// TIA Portal V16 program export: 3 tag tables, 15 data types, 4 data blocks, 30 code blocks (in call order from the OBs), 9 instance data blocks

VAR_GLOBAL   // PLC tag table "Default tag table"
   System_Byte AT %MB1 : Byte;
   FirstScan AT %M1.0 : Bool;
   DiagStatusUpdate AT %M1.1 : Bool;
   AlwaysTRUE AT %M1.2 : Bool;
   AlwaysFALSE AT %M1.3 : Bool;
   Clock_Byte AT %MB0 : Byte;
   Clock_10Hz AT %M0.0 : Bool;
   Clock_5Hz AT %M0.1 : Bool;
   "Clock_2.5Hz" AT %M0.2 : Bool;
   Clock_2Hz AT %M0.3 : Bool;
   "Clock_1.25Hz" AT %M0.4 : Bool;
   Clock_1Hz AT %M0.5 : Bool;
   "Clock_0.625Hz" AT %M0.6 : Bool;
   "Clock_0.5Hz" AT %M0.7 : Bool;
   Tag_1 AT %M100.0 : Bool;
   Tag_2 AT %MW200 : Int;
   Tag_3 AT %M100.1 : Bool;
   Tag_4 AT %M100.2 : Bool;
   Tag_5 AT %M100.3 : Bool;
   Tag_6 AT %M100.4 : Bool;
   Tag_7 AT %M100.5 : Bool;
   Tag_8 AT %M200.0 : Bool;
   Tag_9 AT %MD300 : Real;
   pulse_high AT %M110.0 : Bool;
END_VAR

VAR_GLOBAL   // PLC tag table "input"
   buttonControlCircuit AT %I0.0 : Bool;   // цепи управления
   buttonStart AT %I0.1 : Bool;   // Старт
   buttonStop AT %I0.2 : Bool;   // Стоп
   buttonAlarmStop AT %I0.3 : Bool;   // Аварийный стоп
   M1_alarmCB AT %I0.4 : Bool;   // М1 - авария автоматического выключателя
   M2_alarmCB AT %I0.5 : Bool;   // М2 - авария автоматического выключателя
   isNormalElectrical AT %I0.6 : Bool;   // Сеть в норме
   sensorOverflowReceiverTable AT %I0.7 : Bool;   // Датчик пересыпа приемного стола
   YP1_ReadyAccept AT %I1.0 : Bool;   // УП1 - готов принять
   YP1_StartDozing AT %I1.1 : Bool;   // УП1 - запуск дозирования
   YP2_ReadyAccept AT %I1.2 : Bool;   // УП2 - готов принять
   YP2_StartDozing AT %I1.3 : Bool;   // УП2 - запуск дозирования
END_VAR

VAR_GLOBAL   // PLC tag table "output"
   lampBlue AT %Q0.0 : Bool;   // Синяя лампа
   lampGreen AT %Q0.1 : Bool;   // Зеленая лампа
   lampRed AT %Q0.2 : Bool;   // Красная лампа
   qOn_ControlCurcuit AT %Q0.3 : Bool;   // включение цепей управления
   Y1q_ReadyDoze AT %Q0.4 : Bool;   // УП1 - доза готова
   Y2q_ReadyDoze AT %Q0.5 : Bool;   // УП2 - доза готова
   Conv1_FRV AT %Q0.6 : Bool;   // Конвейер1 - вперед
   Conv1_REV AT %Q0.7 : Bool;   // Конвейер1 - назад
   Conv2_FRV AT %Q1.0 : Bool;   // Конвейер2 - вперед
   Conv2_REV AT %Q1.1 : Bool;   // Конвейер2 - назад
   qDoor1_open AT %Q8.0 : Bool;   // Лопатка - открыть - 1
   qDoor1_close AT %Q8.1 : Bool;   // Лопатка - закрыть- 1
   qDoor2_open AT %Q8.2 : Bool;   // Лопатка - открыть - 2
   qDoor2_close AT %Q8.3 : Bool;   // Лопатка - закрыть- 2
   qDoor3_open AT %Q8.4 : Bool;   // Лопатка - открыть - 3
   qDoor3_close AT %Q8.5 : Bool;   // Лопатка - закрыть- 3
   qDoor4_open AT %Q8.6 : Bool;   // Лопатка - открыть - 4
   qDoor4_close AT %Q8.7 : Bool;   // Лопатка - закрыть- 4
   qDoor5_open AT %Q9.0 : Bool;   // Лопатка - открыть - 5
   qDoor5_close AT %Q9.1 : Bool;   // Лопатка - закрыть- 5
   qDoor6_open AT %Q9.2 : Bool;   // Лопатка - открыть - 6
   qDoor6_close AT %Q9.3 : Bool;   // Лопатка - закрыть- 6
   qDoor7_open AT %Q9.4 : Bool;   // Лопатка - открыть - 7
   qDoor7_close AT %Q9.5 : Bool;   // Лопатка - закрыть- 7
   qDoor8_open AT %Q9.6 : Bool;   // Лопатка - открыть - 8
   qDoor8_close AT %Q9.7 : Bool;   // Лопатка - закрыть- 8
   qBunker3_leftOpen AT %Q12.0 : Bool;   // Бункер - открыть влево - 3
   qBunker3_leftClose AT %Q12.1 : Bool;   // Бункер - закрыть влево - 3
   qBunker3_rightOpen AT %Q12.2 : Bool;   // Бункер - открыть вправо- 3
   qBunker3_rightClose AT %Q12.3 : Bool;   // Бункер - закрыть вправо- 3
   qBunker4_leftOpen AT %Q12.4 : Bool;   // Бункер - открыть влево - 4
   qBunker4_leftClose AT %Q12.5 : Bool;   // Бункер - закрыть влево - 4
   qBunker4_rightOpen AT %Q12.6 : Bool;   // Бункер - открыть вправо- 4
   qBunker4_rightClose AT %Q12.7 : Bool;   // Бункер - закрыть вправо- 4
   qBunker5_leftOpen AT %Q13.0 : Bool;   // Бункер - открыть влево - 5
   qBunker5_leftClose AT %Q13.1 : Bool;   // Бункер - закрыть влево - 5
   qBunker5_rightOpen AT %Q13.2 : Bool;   // Бункер - открыть вправо- 5
   qBunker5_rightClose AT %Q13.3 : Bool;   // Бункер - закрыть вправо- 5
   qBunker6_leftOpen AT %Q13.4 : Bool;   // Бункер - открыть влево - 6
   qBunker6_leftClose AT %Q13.5 : Bool;   // Бункер - закрыть влево - 6
   qBunker6_rightOpen AT %Q13.6 : Bool;   // Бункер - открыть вправо- 6
   qBunker6_rightClose AT %Q13.7 : Bool;   // Бункер - закрыть вправо- 6
   qBunker7_leftOpen AT %Q14.0 : Bool;   // Бункер - открыть влево - 7
   qBunker7_leftClose AT %Q14.1 : Bool;   // Бункер - закрыть влево - 7
   qBunker7_rightOpen AT %Q14.2 : Bool;   // Бункер - открыть вправо- 7
   qBunker7_rightClose AT %Q14.3 : Bool;   // Бункер - закрыть вправо- 7
   qBunker8_leftOpen AT %Q14.4 : Bool;   // Бункер - открыть влево - 8
   qBunker8_leftClose AT %Q14.5 : Bool;   // Бункер - закрыть влево - 8
   qBunker8_rightOpen AT %Q14.6 : Bool;   // Бункер - открыть вправо- 8
   qBunker8_rightClose AT %Q14.7 : Bool;   // Бункер - закрыть вправо- 8
   qBunker9_leftOpen AT %Q15.0 : Bool;   // Бункер - открыть влево - 9
   qBunker9_leftClose AT %Q15.1 : Bool;   // Бункер - закрыть влево - 9
   qBunker9_rightOpen AT %Q15.2 : Bool;   // Бункер - открыть вправо- 9
   qBunker9_rightClose AT %Q15.3 : Bool;   // Бункер - закрыть вправо- 9
   setVibration AT %QW64 : Int;   // задание уровня вибрации
   qDoor9_open AT %Q10.0 : Bool;   // Лопатка - открыть - 9
   qDoor9_close AT %Q10.1 : Bool;   // Лопатка - закрыть- 9
   qDoor10_open AT %Q10.2 : Bool;   // Лопатка - открыть - 10
   qDoor10_close AT %Q10.3 : Bool;   // Лопатка - закрыть- 10
   qDoor11_open AT %Q10.4 : Bool;   // Лопатка - открыть - 11
   qDoor11_close AT %Q10.5 : Bool;   // Лопатка - закрыть- 11
   qDoor12_open AT %Q10.6 : Bool;   // Лопатка - открыть - 12
   qDoor12_close AT %Q10.7 : Bool;   // Лопатка - закрыть- 12
   qBunker1_leftOpen AT %Q11.0 : Bool;   // Бункер - открыть влево - 1
   qBunker1_leftClose AT %Q11.1 : Bool;   // Бункер - закрыть влево - 1
   qBunker1_rightOpen AT %Q11.2 : Bool;   // Бункер - открыть вправо - 1
   qBunker1_rightClose AT %Q11.3 : Bool;   // Бункер - закрыть вправо - 1
   qBunker2_leftOpen AT %Q11.4 : Bool;   // Бункер - открыть влево - 2
   qBunker2_leftClose AT %Q11.5 : Bool;   // Бункер - закрыть влево - 2
   qBunker2_rightOpen AT %Q11.6 : Bool;   // Бункер - открыть вправо - 2
   qBunker2_rightClose AT %Q11.7 : Bool;   // Бункер - закрыть вправо - 2
   qBunker11_leftOpen AT %Q16.0 : Bool;   // Бункер - открыть влево - 11
   qBunker11_leftClose AT %Q16.1 : Bool;   // Бункер - закрыть влево - 11
   qBunker11_rightOpen AT %Q16.2 : Bool;   // Бункер - открыть вправо- 11
   qBunker11_rightClose AT %Q16.3 : Bool;   // Бункер - закрыть вправо- 11
   qBunker12_leftOpen AT %Q16.4 : Bool;   // Бункер - открыть влево - 12
   qBunker12_leftClose AT %Q16.5 : Bool;   // Бункер - закрыть влево - 12
   qBunker12_rightOpen AT %Q16.6 : Bool;   // Бункер - открыть вправо- 12
   qBunker12_rightClose AT %Q16.7 : Bool;   // Бункер - закрыть вправо- 12
   qBunker10_leftOpen AT %Q15.4 : Bool;   // Бункер - открыть влево - 10
   qBunker10_leftClose AT %Q15.5 : Bool;   // Бункер - закрыть влево - 10
   qBunker10_rightOpen AT %Q15.6 : Bool;   // Бункер - открыть вправо- 10
   qBunker10_rightClose AT %Q15.7 : Bool;   // Бункер - закрыть вправо- 10
   qFlipperUp AT %Q17.0 : Bool;   // плавник поднять
   qFlipperDown AT %Q17.1 : Bool;   // плавник опустить
   qVibroLot7_On AT %Q18.2 : Bool;   // управление вибролотком 7
   qVibroLot8_On AT %Q18.3 : Bool;   // управление вибролотком 8
   qVibroLot9_On AT %Q18.4 : Bool;   // управление вибролотком 9
   qVibroLot10_On AT %Q18.5 : Bool;   // управление вибролотком 10
   qVibroLot11_On AT %Q18.6 : Bool;   // управление вибролотком 11
   qVibroLot12_On AT %Q18.7 : Bool;   // управление вибролотком 12
   qVibroLot6_On AT %Q18.1 : Bool;   // управление вибролотком 6
   qVibroLot5_On AT %Q18.0 : Bool;   // управление вибролотком 5
   qVibroLot1_On AT %Q17.4 : Bool;   // управление вибролотком 1
   qVibroLot2_On AT %Q17.5 : Bool;   // управление вибролотком 2
   qVibroLot3_On AT %Q17.6 : Bool;   // управление вибролотком 3
   qVibroLot4_On AT %Q17.7 : Bool;   // управление вибролотком 4
   qVibroTable1 AT %Q17.2 : Bool;   // управление вибростолом 1
   qVibrotable2 AT %Q17.3 : Bool;   // управление вибростолом 2
   setSpeedConv AT %QW66 : Int;   // задание скорости конвейера
   startSourceConveyer AT %Q19.0 : Bool;   // запуск питателя
END_VAR

TYPE "LineWeight"
// stored: IsFailsafeCompliant false
   STRUCT
      isVibroLotWork : Bool;   // работа вибролотка
      percentVibroLot : Int;   // текущая вибрация вибролотка
      stateValveAfterVibroLot : Bool;   // состояние закрылки после вибролотка
      stateLeftValveWeightPocket : Bool;   // состояние левого клапана открывающегося кармана
      stateRightValveWeightPocket : Bool;   // состояние правого клапана открывающегося кармана
      targetWeightPocket : Real;   // целевой вес кармана
      currentWeightPocket : Real;   // текущий вес в кармане
      manOpenValveAfterVibroLot : Bool;   // ручн - открыть лопатку
      manCloseValveAfterVibroLot : Bool;   // ручн - закрыть лопатку
      manOpenLeftValveWeightPocket : Bool;   // ручн -открыть левый карман
      manCloseLeftValveWeightPocket : Bool;   // ручн -закрыть левый карман
      manOpenRightValveWeightPocket : Bool;   // ручн - открыть правый карман
      manCloseRightValveWieghtPocket : Bool;   // ручн - закрыть правый карман
      manVibroLotStart : Bool;   // ручн - управление ПУСК\Стоп вибролотка
      begWeightModuleReady : Bool;   // начальный экран - готовность весоизмерительного модуля
   END_STRUCT;
END_TYPE

TYPE "ReadyWeight"
// stored: IsFailsafeCompliant false
   STRUCT
      ready1Machine : Bool;
      ready2Machine : Bool;
   END_STRUCT;
END_TYPE

TYPE "addedVibro"
// stored: IsFailsafeCompliant false
   STRUCT
      manStartVibroTable : Array[0..2] of Bool;   // запуск вибростола в ручном режиме
      manValueVibro : Int;   // величина вибрации в ручном режиме
      stateVibroTable : Array[0..2] of Bool;
   END_STRUCT;
END_TYPE

TYPE "alarmsPlant"
// stored: IsFailsafeCompliant false
   STRUCT
      bit : Array[0..83] of Bool;
   END_STRUCT;
END_TYPE

TYPE "calibrationModule"
// stored: IsFailsafeCompliant false
   STRUCT
      calib : Array[0..12] of Bool;
      tara : Array[0..12] of Bool;
      valReadyWModule : Int;   // +- величина готовности модуля
   END_STRUCT;
END_TYPE

TYPE "cleaningMode"
// stored: IsFailsafeCompliant false
   STRUCT
      allWeightModuleReady : Bool;   // Все весоизмерительные модули готовы
      pauseClean : Bool;   // пауза очистки
      progressClean : Int;   // прогресс очистки
      runClean : Bool;   // запуск очистки
      timeClean : Int;   // время очистки
   END_STRUCT;
END_TYPE

TYPE "dataStantion"
// stored: IsFailsafeCompliant false
   STRUCT
      numberDozInMin : Int;   // число доз в минуту
      numberDozInthisWeight : Int;   // полученное число доз заданной порции
      nuvberDozSmena : Int;   // число доз за смену
      currentPogreshn1 : Real;   // погрешность для текущей дозы 1 машины
      currentPogr2 : Real;   // погрешность для текущей дозы 2 машины
      maxPogr : Real;   // максимальная погрешность для порции
      isEmulation : Bool;
      emulStartDozing : Array[0..2] of Bool;
      emulReadyAccept : Array[0..2] of Bool;
   END_STRUCT;
END_TYPE

TYPE "dateTime"
// stored: IsFailsafeCompliant false
   STRUCT
      year : Int;
      month : Int;
      day : Int;
      hour : Int;
      minute : Int;
      second : Int;
   END_STRUCT;
END_TYPE

TYPE "mode"
// stored: IsFailsafeCompliant false
   STRUCT
      Yq_ReadyDoze : Array[0..2] of Bool;
      Conv_FRV : Array[0..2] of Bool;   // Конвейер1 - вперед
      Conv_REV : Array[0..2] of Bool;   // Конвейер1 - назад
      Door_open : Array[0..12] of Bool;   // Лопатка - открыть
      Door_close : Array[0..12] of Bool;   // Лопатка - закрыть
      Bunker_leftOpen : Array[0..12] of Bool;   // Бункер - открыть влево
      Bunker_leftClose : Array[0..12] of Bool;   // Бункер - закрыть влево
      Bunker_rightOpen : Array[0..12] of Bool;   // Бункер - открыть вправо
      Bunker_rightClose : Array[0..12] of Bool;   // Бункер - закрыть вправо
      flipper_Up : Bool;   // управление плавником вверх
      flipper_Down : Bool;   // управление плавником вниз
      vibroTable : Array[0..2] of Bool;   // управление вибростолом
      vibroLot : Array[0..12] of Bool;   // управление вибролотком
      setVibration : Real;   // уставка вибрации
      setSpeedInConv : Real;   // скорость питателя
      startInConv : Bool;   // запуск питателя
   END_STRUCT;
END_TYPE

TYPE "outConv"
// stored: IsFailsafeCompliant false
   STRUCT
      isUpInBegin : Bool;   // направление вращения для упаковки
      isUseInBegin : Bool;   // использовать ли конвейер для упаковки
      isUpInEnd : Bool;   // направления вращения при очистке
      setWeightPack : Real;   // вес упаковки
      currentWeightPack : Real;   // текущий вес упаковки
      currentErrorMeasure : Real;   // текущая погрешность
      isWorkConv : Bool;   // работа конвейера
      isAlarmConv : Bool;   // авария конвейера
      isReadyPackingMachine : Bool;   // сигнал готовности упаковочной машины
      isReadyDozaPackingMachine : Bool;   // сигнал доза упаковочной машины
      manStartOutConv : Bool;   // ручн - запуск конвейера
      stateConvInt : Int;   // состояние конвейера
      manIsUpConv : Bool;   // ручн - конв вперед\назад
   END_STRUCT;
END_TYPE

TYPE "plavnik"
// stored: IsFailsafeCompliant false
   STRUCT
      statePlavnik : Bool;   // состояние плавника
      manOpenPlavnik : Bool;   // ручн - открытие клапана
      manClosePlavnik : Bool;   // ручн - закрытие клапана
   END_STRUCT;
END_TYPE

TYPE "recipeVar"
// stored: IsFailsafeCompliant false
   STRUCT
      setWeight : Real;   // весовая уставка в рецепте
      speed_InConveyer : Int;   // скорость конвейера питателя( конвейер на входе системы)
      speedVibro : Int;   // скорость вибролотков(одна на все)
      maxWeightBunker : Real;   // максимальный вес бункеров
      workPlavnik : Bool;   // работа плавника
      measurmentError : Real;   // допускаемая погрешность веса в общем сбросе
      mediumWeightProduct : Real;   // средний вес продукта
   END_STRUCT;
END_TYPE

TYPE "rotary"
// stored: IsFailsafeCompliant false
   STRUCT
      rotUp1 : Int;
      rotDown1 : Int;
      rotUp2 : Int;
      rotDown2 : Int;
   END_STRUCT;
END_TYPE

TYPE "sourceConv"
// stored: IsFailsafeCompliant false
   STRUCT
      currentSpeed : Int;   // ОС скорость
      manSetSpeed : Int;   // ручн - задание скорости
      isConvWork : Bool;   // конв работает
      isConvAlarm : Bool;   // авария конв
      manStartConv : Bool;   // ручн - старт конвейера
      stateConvInt : Int;   // состояние конвейера
      setSpeedWeightLimit : Int;   // скорость питателя при перевесе
   END_STRUCT;
END_TYPE

TYPE "stableWeight"
// stored: IsFailsafeCompliant false
   STRUCT
      weight : Array[0..10] of Real;
   END_STRUCT;
END_TYPE

DATA_BLOCK "IO"   // DB10
{ S7_Optimized_Access := 'TRUE' }
VERSION : 0.1
// stored: AutoNumber false, DBAccessibleFromOPCUA true, IsOnlyStoredInLoadMemory false, IsRetainMemResEnabled false, IsWriteProtectedInAS false, MemoryReserve 100
   VAR
      input : Struct
         buttonControlCircuit : Bool;   // цепи управления
         buttonStart : Bool;   // Старт
         buttonStop : Bool;   // Стоп
         buttonAlarmStop : Bool;   // Аварийный стоп
         M_alarmCB : Array[0..2] of Bool;   // М - авария автоматического выключателя
         isNormalElectrical : Bool;   // Сеть в норме
         sensorOverflowReceiverTable : Bool;   // Датчик пересыпа приемного стола
         YP_ReadyAccept : Array[0..2] of Bool;   // УП - готов принять
         YP_StartDozing : Array[0..2] of Bool;   // УП - запуск дозирования
      END_STRUCT;
      output : Struct
         lampBlue : Bool;   // Синяя лампа
         lampGreen : Bool;   // Зеленая лампа
         lampRed : Bool;   // Красная лампа
         qOn_ControlCurcuit : Bool;   // включение цепей управления
         Yq_ReadyDoze : Array[0..2] of Bool;   // УП - доза готова
         Conv_FRV : Array[0..2] of Bool;   // Конвейер1 - вперед
         Conv_REV : Array[0..2] of Bool;   // Конвейер1 - назад
         Door_open : Array[0..12] of Bool;   // Лопатка - открыть
         Door_close : Array[0..12] of Bool;   // Лопатка - закрыть
         Bunker_leftOpen : Array[0..12] of Bool;   // Бункер - открыть влево
         Bunker_leftClose : Array[0..12] of Bool;   // Бункер - закрыть влево
         Bunker_rightOpen : Array[0..12] of Bool;   // Бункер - открыть вправо
         Bunker_rightClose : Array[0..12] of Bool;   // Бункер - закрыть вправо
         flipper_Up : Bool;   // управление плавником вверх
         flipper_Down : Bool;   // управление плавником вниз
         vibroTable : Array[0..2] of Bool;   // управление вибростолом
         vibroLot : Array[0..12] of Bool;   // управление вибролотком
         setVibration : Real;   // уставка вибрации
         setSpeed : Real;   // уставка скорости конвейера
         convSource : Bool;   // запуск питателя
      END_STRUCT;
   END_VAR
BEGIN
END_DATA_BLOCK

DATA_BLOCK "hmi"   // DB200
{ S7_Optimized_Access := 'FALSE' }
VERSION : 0.1
// stored: AutoNumber false, DBAccessibleFromOPCUA true, IsOnlyStoredInLoadMemory false, IsWriteProtectedInAS false
   VAR
      alarmTest : "alarmsPlant";
      autoMode : Bool;   // автоматический режим
      isEnableAutoMode : Bool;
      calibrWeightMode : "calibrationModule";   // калибровка и тарирование весов
      dataStantion : "dataStantion";
      manRunAllVibroLot : Bool;
      manStopAllVibroLot : Bool;
      NewReadyWeightOnLine : Array[0..12] of Bool;
      outConvAndPack : Array[0..2] of "outConv";
      permitOn1Bunk : Array[0..12] of Bool;
      permitOn2Bunk : Array[0..12] of Bool;
      plavnik : "plavnik";
      readySystem : Int;
      recipeVar : "recipeVar";   // переменные рецепта
      rotary : "rotary";   // анимация вращения конвейеров
      sourceConv : "sourceConv";
      timeWorkConvAuto : Int;
      weightLine : Array[0..12] of "LineWeight";
      currentSetRecipes : String := '$00$00';
      numPage : Int;
      commonAlarm : Bool;   // Сигнал если хотябы одна авария есть
      report : Struct
         perfomance : Int;   // производительность
         sumPreWeight : Real;   // суммарная переработка веса
         commonTimeWork : Real;   // время работы установки
      END_STRUCT;
      addedVibro : "addedVibro";
   END_VAR
BEGIN
   // alarmTest.bit[0] : Управляющие цепи деактивированны
   // alarmTest.bit[1] : весовой модуль не в сети 1
   // alarmTest.bit[2] : весовой модуль не в сети 2
   // alarmTest.bit[3] : весовой модуль не в сети 3
   // alarmTest.bit[4] : весовой модуль не в сети 4
   // alarmTest.bit[5] : весовой модуль не в сети 5
   // alarmTest.bit[6] : весовой модуль не в сети 6
   // alarmTest.bit[7] : весовой модуль не в сети 7
   // alarmTest.bit[8] : весовой модуль не в сети 8
   // alarmTest.bit[9] : весовой модуль не в сети 9
   // alarmTest.bit[10] : весовой модуль не в сети 10
   // alarmTest.bit[11] : весовой модуль не в сети 11
   // alarmTest.bit[12] : весовой модуль не в сети 12
   // alarmTest.bit[13] : обрыв датчик весового модуля 1 -значение выше 7000
   // alarmTest.bit[14] : обрыв датчик весового модуля 2
   // alarmTest.bit[15] : обрыв датчик весового модуля 3
   // alarmTest.bit[16] : обрыв датчик весового модуля 4
   // alarmTest.bit[17] : обрыв датчик весового модуля 5
   // alarmTest.bit[18] : обрыв датчик весового модуля 6
   // alarmTest.bit[19] : обрыв датчик весового модуля 7
   // alarmTest.bit[20] : обрыв датчик весового модуля 8
   // alarmTest.bit[21] : обрыв датчик весового модуля 9
   // alarmTest.bit[22] : обрыв датчик весового модуля 10
   // alarmTest.bit[23] : обрыв датчик весового модуля 11
   // alarmTest.bit[24] : обрыв датчик весового модуля 12
   // alarmTest.bit[25] : Напряжение сети не в норме
   // alarmTest.bit[26] : Тепловое реле Конв1
   // alarmTest.bit[27] : тепловое реле Конв2
   // alarmTest.bit[58] : Нажат аварийный пост
   // alarmTest.bit[59] : Авария бункер 1
   // alarmTest.bit[60] : Авария бункер 2
   // alarmTest.bit[61] : Авария бункер 3
   // alarmTest.bit[62] : Авария бункер 4
   // alarmTest.bit[63] : Авария бункер 5
   // alarmTest.bit[64] : Авария бункер 6
   // alarmTest.bit[65] : Авария бункер 7
   // alarmTest.bit[66] : Авария бункер 8
   // alarmTest.bit[67] : Авария бункер 9
   // alarmTest.bit[68] : Авария бункер 10
   // alarmTest.bit[69] : Авария бункер 11
   // alarmTest.bit[70] : Авария бункер 12
   // alarmTest.bit[83] : Нет возможности сформировать порцию
   // calibrWeightMode.calib : калибровка весов
   // calibrWeightMode.tara : тарирование весов
END_DATA_BLOCK

DATA_BLOCK "signalKVSStation"   // DB20
{ S7_Optimized_Access := 'TRUE' }
VERSION : 0.1
// stored: AutoNumber false, DBAccessibleFromOPCUA true, IsOnlyStoredInLoadMemory false, IsRetainMemResEnabled false, IsWriteProtectedInAS false, MemoryReserve 100
   VAR
      isWorkControlCircuit : Bool;   // цепи управления активированы
      isStopAlarm : Bool;   // приход любой аварии которая останавливает установку
      isOtherAlarm : Bool;   // приход просто аварий
      isStartAutoMode : Bool;   // начало работы в автоматическом режиме
      enableAutoMode : Bool;   // разрешение перевода в автоматический режим
      isPreparationAutoModeFinish : Bool;   // подготовк к запуску автоматического режима
      enableManualMode : Bool;   // разрешение работы в ручном режиме
      qManualMode : "mode";   // активация катушек в ручном режиме
      qAutoMode : "mode";   // активация катушек в автоматическом режиме
      currentWeight : Array[0..12] of Real;   // вес получаемый по модбасу
      stableWeight : Array[0..12] of "stableWeight";   // установившийся вес в бункерах
   END_VAR
BEGIN
END_DATA_BLOCK

DATA_BLOCK "bufferModBus"   // DB4
{ S7_Optimized_Access := 'FALSE' }
VERSION : 0.1
// stored: AutoNumber true, DBAccessibleFromOPCUA true, IsOnlyStoredInLoadMemory false, IsWriteProtectedInAS false
   VAR
      Buffer_DataModbusPort1 { ExternalAccessible := 'False'; ExternalVisible := 'False'; ExternalWritable := 'False'} : Array[0..20] of Word;
      Buffer_DataModbusPort2 { ExternalAccessible := 'False'; ExternalVisible := 'False'; ExternalWritable := 'False'} : Array[0..20] of Word;
   END_VAR
BEGIN
END_DATA_BLOCK

ORGANIZATION_BLOCK "Main"   // OB1, LAD, ProgramCycle
TITLE = "Main Program Sweep (Cycle)"
{ S7_Optimized_Access := 'TRUE' }
VERSION : 0.1
// stored: AutoNumber true, IsIECCheckEnabled false, SetENOAutomatically false
   VAR_INPUT
      Initial_Call : Bool;   // Initial call of this OB
      Remanence : Bool;   // =True, if remanent data are available
   END_VAR
BEGIN

REGION Network 1: опрос весов
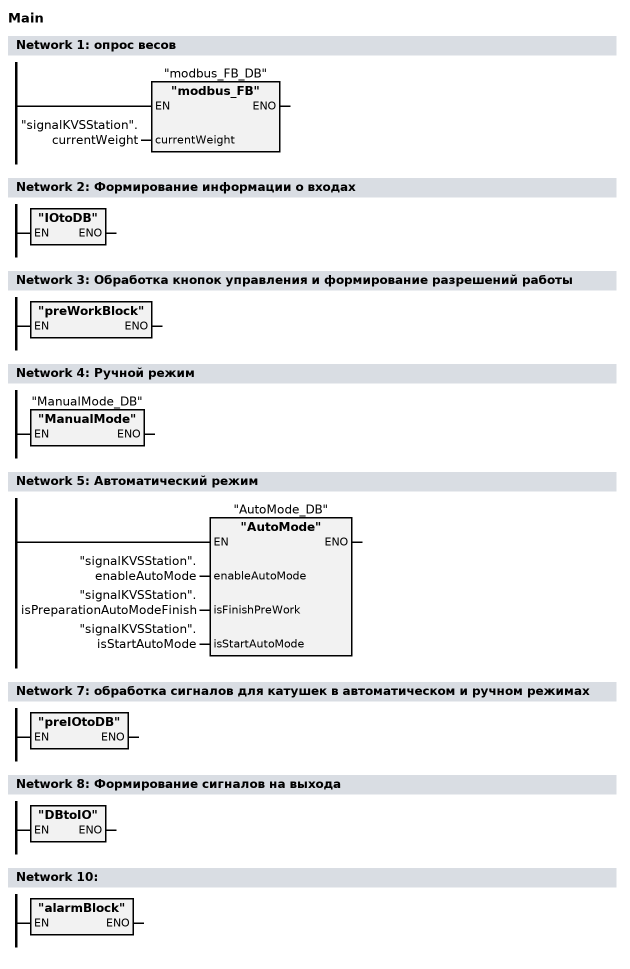
   RUNG wire#powerrail
      "modbus_FB_DB"(currentWeight := "signalKVSStation".currentWeight)
   END_RUNG
   // the same network as SCL:
   "modbus_FB_DB"(currentWeight := "signalKVSStation".currentWeight);   // "modbus_FB"
END_REGION

REGION Network 2: Формирование информации о входах
   RUNG wire#powerrail
      "IOtoDB"()
   END_RUNG
   // the same network as SCL:
   "IOtoDB"();
END_REGION

REGION Network 3: Обработка кнопок управления и формирование разрешений работы
   RUNG wire#powerrail
      "preWorkBlock"()
   END_RUNG
   // the same network as SCL:
   "preWorkBlock"();
END_REGION

REGION Network 4: Ручной режим
   RUNG wire#powerrail
      "ManualMode_DB"()
   END_RUNG
   // the same network as SCL:
   "ManualMode_DB"();   // "ManualMode"
END_REGION

REGION Network 5: Автоматический режим
   RUNG wire#powerrail
      "AutoMode_DB"(enableAutoMode := "signalKVSStation".enableAutoMode, isFinishPreWork := "signalKVSStation".isPreparationAutoModeFinish, isStartAutoMode := "signalKVSStation".isStartAutoMode)
   END_RUNG
   // the same network as SCL:
   "AutoMode_DB"(enableAutoMode := "signalKVSStation".enableAutoMode,   // "AutoMode"
                 isFinishPreWork := "signalKVSStation".isPreparationAutoModeFinish,
                 isStartAutoMode := "signalKVSStation".isStartAutoMode);
END_REGION

REGION Network 7: обработка сигналов для катушек в автоматическом и ручном режимах
   RUNG wire#powerrail
      "preIOtoDB"()
   END_RUNG
   // the same network as SCL:
   "preIOtoDB"();
END_REGION

REGION Network 8: Формирование сигналов на выхода
   RUNG wire#powerrail
      "DBtoIO"()
   END_RUNG
   // the same network as SCL:
   "DBtoIO"();
END_REGION

REGION Network 10
   RUNG wire#powerrail
      "alarmBlock"()
   END_RUNG
   // the same network as SCL:
   "alarmBlock"();
END_REGION
END_ORGANIZATION_BLOCK

FUNCTION_BLOCK "modbus_FB"   // FB9, LAD
{ S7_Optimized_Access := 'TRUE' }
VERSION : 0.1
// stored: AutoNumber true, IsIECCheckEnabled false, IsRetainMemResEnabled false, MemoryReserve 100, SetENOAutomatically false, UDAEnableTagReadback false
   VAR_IN_OUT
      currentWeight : Array[0..12] of Real;
   END_VAR
   VAR
      MODBUS_ADDRESS : Array[0..12] of UInt;
      modbus_SenecaConnectPort1_FB : "modbus_SenecaConnectPort1";
      modbus_SenecaConnectPort2_FB : "modbus_SenecaConnectPort2";
   END_VAR
   VAR_TEMP
      i : SInt;
   END_VAR
   // MODBUS_ADDRESS[1] := 10;
   // MODBUS_ADDRESS[2] := 11;
   // MODBUS_ADDRESS[3] := 12;
   // MODBUS_ADDRESS[4] := 13;
   // MODBUS_ADDRESS[5] := 14;
   // MODBUS_ADDRESS[6] := 15;
   // MODBUS_ADDRESS[7] := 20;
   // MODBUS_ADDRESS[8] := 21;
   // MODBUS_ADDRESS[9] := 22;
   // MODBUS_ADDRESS[10] := 23;
   // MODBUS_ADDRESS[11] := 24;
   // MODBUS_ADDRESS[12] := 25;
BEGIN

REGION Network 1: ОПРОС МОДУЛЕЙ ЧЕРЕРЗ 1 ПОРТ
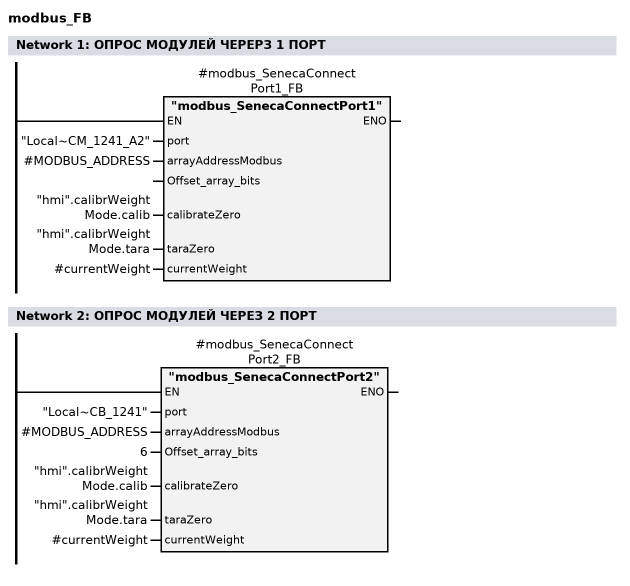
   RUNG wire#powerrail
      #modbus_SenecaConnectPort1_FB(port := "Local~CM_1241_A2", arrayAddressModbus := #MODBUS_ADDRESS, Offset_array_bits :=, calibrateZero := "hmi".calibrWeightMode.calib, taraZero := "hmi".calibrWeightMode.tara, currentWeight := #currentWeight)
   END_RUNG
   // the same network as SCL:
   #modbus_SenecaConnectPort1_FB(port := "Local~CM_1241_A2",   // "modbus_SenecaConnectPort1"
                           arrayAddressModbus := #MODBUS_ADDRESS,
                           calibrateZero := "hmi".calibrWeightMode.calib,
                           taraZero := "hmi".calibrWeightMode.tara,
                           currentWeight := #currentWeight);
END_REGION

REGION Network 2: ОПРОС МОДУЛЕЙ ЧЕРЕЗ 2 ПОРТ
   RUNG wire#powerrail
      #modbus_SenecaConnectPort2_FB(port := "Local~CB_1241", arrayAddressModbus := #MODBUS_ADDRESS, Offset_array_bits := 6, calibrateZero := "hmi".calibrWeightMode.calib, taraZero := "hmi".calibrWeightMode.tara, currentWeight := #currentWeight)
   END_RUNG
   // the same network as SCL:
   #modbus_SenecaConnectPort2_FB(port := "Local~CB_1241",   // "modbus_SenecaConnectPort2"
                           arrayAddressModbus := #MODBUS_ADDRESS,
                           Offset_array_bits := 6,
                           calibrateZero := "hmi".calibrWeightMode.calib,
                           taraZero := "hmi".calibrWeightMode.tara,
                           currentWeight := #currentWeight);
END_REGION

REGION Network 3 (SCL): Передаем вес в панель
   #i := 0;
   FOR #i := 1 TO 12 DO
       "hmi".weightLine[#i].currentWeightPocket := #currentWeight[#i];
   END_FOR;
END_REGION

REGION Network 4 (SCL)
   IF "hmi".calibrWeightMode.tara[0] THEN
       #i := 0;
       FOR #i := 1 TO 12 DO
           "hmi".calibrWeightMode.tara[#i] := true;
       END_FOR;
   END_IF;
END_REGION
END_FUNCTION_BLOCK

FUNCTION_BLOCK "modbus_SenecaConnectPort1"   // FB11, LAD
{ S7_Optimized_Access := 'TRUE' }
VERSION : 0.1
// stored: AutoNumber true, IsIECCheckEnabled false, IsRetainMemResEnabled false, MemoryReserve 100, SetENOAutomatically false, UDAEnableTagReadback false
   VAR_INPUT
      port : PORT;   // порт для подключения
      arrayAddressModbus : Array[0..12] of UInt;
      Offset_array_bits : SInt;
   END_VAR
   VAR_IN_OUT
      calibrateZero : Array[0..12] of Bool;
      taraZero : Array[0..12] of Bool;
      currentWeight : Array[0..12] of Real;
   END_VAR
   VAR
      MB_COMM_LOAD : MB_COMM_LOAD;
      MB_MASTER : MB_MASTER;
      Data_toMB_MASTER : Struct
         REQ : Bool;
         MB_ADDR : UInt;
         MODE : USInt;
         DATA_ADDR : UDInt;
         DATA_LEN : UInt;
         DONE : Bool;
         BUSY : Bool;
         ERROR : Bool;
      END_STRUCT;
      Seneca : Struct
         TON_changeStep : TON_TIME;
         TON_Start { S7_SetPoint := 'True'} : Bool;
         "Step" : SInt;
      END_STRUCT;
      tmpWeight : Array[0..12] of DWord;
      restartPort : Bool;   // перезагрузка Modbus
   END_VAR
   VAR_TEMP
      index : DInt;
      tmpIndex : DInt;
   END_VAR
   // MB_COMM_LOAD.RESP_TO := 100;
   VAR_TEMP   // added for the SCL form of the ladder/FBD networks
      _w1 : Bool;
   END_VAR
BEGIN

REGION Network 1: ИНИЦИАЛИЗИРУЕМ ПОРТ
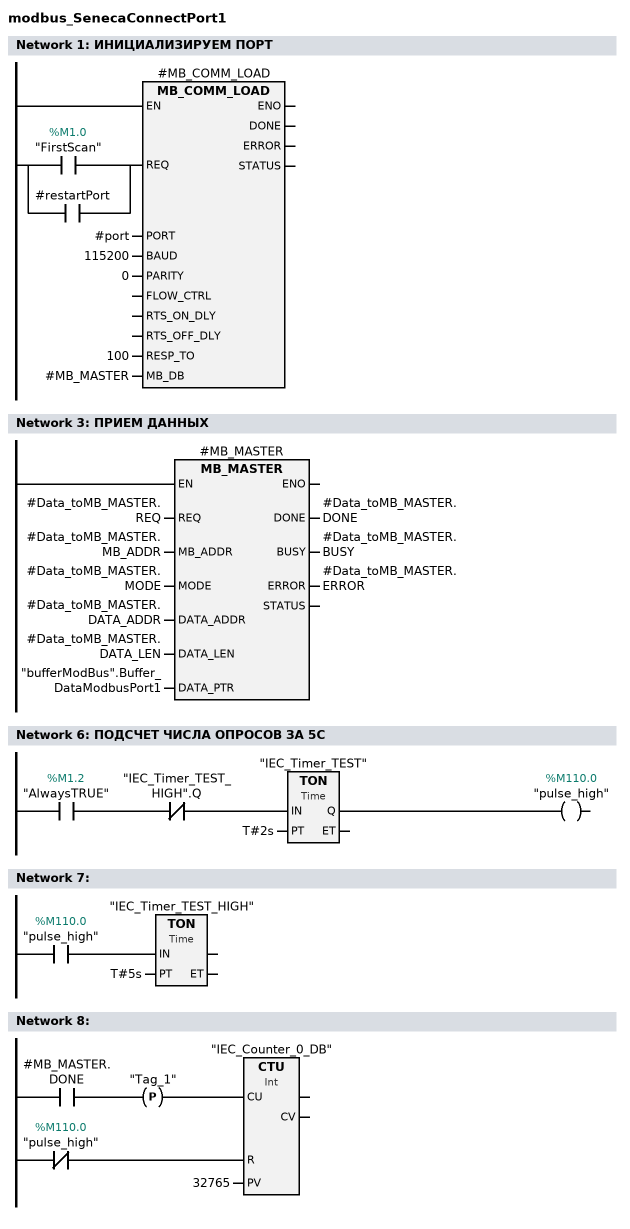
   RUNG wire#powerrail
      #MB_COMM_LOAD.MB_COMM_LOAD(REQ := wire#w1, PORT := #port, BAUD := 115200, PARITY := 0, FLOW_CTRL :=, RTS_ON_DLY :=, RTS_OFF_DLY :=, RESP_TO := 100, MB_DB := #MB_MASTER, DONE =>, ERROR =>, STATUS =>)
   END_RUNG
   RUNG wire#powerrail
      Contact( "FirstScan" )
   END_RUNG wire#w1
   RUNG wire#powerrail
      Contact( #restartPort )
   END_RUNG wire#w1
   // the same network as SCL:
   #MB_COMM_LOAD(REQ := "FirstScan" OR #restartPort,   // MB_COMM_LOAD
                 PORT := #port,
                 BAUD := 115200,
                 PARITY := 0,
                 RESP_TO := 100,
                 MB_DB := #MB_MASTER);
END_REGION

REGION Network 2 (SCL): ОБМЕН
   #Seneca.TON_changeStep(IN :=#Seneca.TON_Start,
                          PT := t#30ms);

   CASE #Seneca.Step OF

       1:
           #Seneca.Step := #Seneca.Step + 1;

       2: //ЧИТАЕМ ЗНАЧЕНИЕ ВЕСА С ПЕРВОГО МОДУЛЯ

           #index := 1+#Offset_array_bits;//заполнять функцию будем через индекс чтобы меньше писать
           "rcvDataWeight"(ADDR_DEVICE := #arrayAddressModbus[#index],
                           Ton_changeStep:=#Seneca.TON_changeStep.Q,
                           Ton_Start:=#Seneca.TON_Start,
                           "Step":=#Seneca.Step,
                           MB_MASTER:=#Data_toMB_MASTER);

       3://ЧИТАЕМ ЗНАЧЕНИЕ ВЕСА СО ВТОРОГО МОДУЛЯ
           #index := 2+#Offset_array_bits;//заполнять функцию будем через индекс чтобы меньше писать
           "rcvDataWeight"(ADDR_DEVICE := #arrayAddressModbus[#index],
                           Ton_changeStep:=#Seneca.TON_changeStep.Q,
                           Ton_Start:=#Seneca.TON_Start,
                           "Step":=#Seneca.Step,
                           MB_MASTER:=#Data_toMB_MASTER);

       4: // КАЛИБРОВКА 0 ДЛЯ ПЕРВОГО МОДУЛЯ и ТАРИРОВАНИЕ
           #index := 1+#Offset_array_bits;//заполнять функцию будем через индекс чтобы меньше писать
           "sndCALIBR&Tara"(ADDR_DEVICE := #arrayAddressModbus[#index],
                        ton_changeStep:=#Seneca.TON_changeStep.Q,
                        MB_MASTER:=#Data_toMB_MASTER,
                        Ton_Start:=#Seneca.TON_Start,
                        Calibrate:=#calibrateZero[#index],
                        Buffer:="bufferModBus".Buffer_DataModbusPort1,
                        "Step":=#Seneca.Step,
                        Tara:=#taraZero[#index]);


       5:// КАЛИБРОВКА 0 ДЛЯ ВТОРОГО МОДУЛЯ и ТАРИРОВАНИЕ
           #index := 2+#Offset_array_bits;//заполнять функцию будем через индекс чтобы меньше писать
           "sndCALIBR&Tara"(ADDR_DEVICE := #arrayAddressModbus[#index],
                        ton_changeStep := #Seneca.TON_changeStep.Q,
                        MB_MASTER := #Data_toMB_MASTER,
                        Ton_Start := #Seneca.TON_Start,
                        Calibrate := #calibrateZero[#index],
                        Buffer := "bufferModBus".Buffer_DataModbusPort1,
                        "Step" := #Seneca.Step,
                        Tara := #taraZero[#index]);

           //////////////////////////////////////////////////////////////////////////////////
           //////////////////////////////////////////////////////////////////////////////////
           //////////////////////////////////////////////////////////////////////////////////
           //////////////////////////////////////////////////////////////////////////////////
       6: //ЧИТАЕМ ЗНАЧЕНИЕ ВЕСА С ТРЕТЬЕГО МОДУЛЯ

           #index := 3+#Offset_array_bits;//заполнять функцию будем через индекс чтобы меньше писать
           "rcvDataWeight"(ADDR_DEVICE := #arrayAddressModbus[#index],
                           Ton_changeStep := #Seneca.TON_changeStep.Q,
                           Ton_Start := #Seneca.TON_Start,
                           "Step" := #Seneca.Step,
                           MB_MASTER := #Data_toMB_MASTER);

       7://ЧИТАЕМ ЗНАЧЕНИЕ ВЕСА С ЧЕТВЕРТОГО МОДУЛЯ
           #index := 4+#Offset_array_bits;//заполнять функцию будем через индекс чтобы меньше писать
           "rcvDataWeight"(ADDR_DEVICE := #arrayAddressModbus[#index],
                           Ton_changeStep := #Seneca.TON_changeStep.Q,
                           Ton_Start := #Seneca.TON_Start,
                           "Step" := #Seneca.Step,
                           MB_MASTER := #Data_toMB_MASTER);

       8:// КАЛИБРОВКА 0 ДЛЯ ТРЕТЬЕГО  МОДУЛЯ

           #index := 3+#Offset_array_bits;//заполнять функцию будем через индекс чтобы меньше писать
           "sndCALIBR&Tara"(ADDR_DEVICE := #arrayAddressModbus[#index],
                        ton_changeStep := #Seneca.TON_changeStep.Q,
                        MB_MASTER := #Data_toMB_MASTER,
                        Ton_Start := #Seneca.TON_Start,
                        Calibrate := #calibrateZero[#index],
                        Buffer := "bufferModBus".Buffer_DataModbusPort1,
                        "Step" := #Seneca.Step,
                        Tara := #taraZero[#index]);

       9://КАЛИБРОВКА 0 ДЛЯ ЧЕТВЕРТОГО МОДУЛЯ

           #index := 4+#Offset_array_bits;//заполнять функцию будем через индекс чтобы меньше писать
           "sndCALIBR&Tara"(ADDR_DEVICE := #arrayAddressModbus[#index],
                        ton_changeStep := #Seneca.TON_changeStep.Q,
                        MB_MASTER := #Data_toMB_MASTER,
                        Ton_Start := #Seneca.TON_Start,
                        Calibrate := #calibrateZero[#index],
                        Buffer := "bufferModBus".Buffer_DataModbusPort1,
                        "Step" := #Seneca.Step,
                        Tara := #taraZero[#index]);

           /////////////////////////////////////////////////////////////////////////////////
           ////////////////////////////////////////////////////////////////////////////////
           ////////////////////////////////////////////////////////////////////////////////
           ////////////////////////////////////////////////////////////////////////////////
       10: //ЧИТАЕМ ЗНАЧЕНИЕ ВЕСА С ПЯТОГО МОДУЛЯ
           #index := 5+#Offset_array_bits;//заполнять функцию будем через индекс чтобы меньше писать
           "rcvDataWeight"(ADDR_DEVICE := #arrayAddressModbus[#index],
                           Ton_changeStep := #Seneca.TON_changeStep.Q,
                           Ton_Start := #Seneca.TON_Start,
                           "Step" := #Seneca.Step,
                           MB_MASTER := #Data_toMB_MASTER);

       11://ЧИТАЕМ ЗНАЧЕНИЕ ВЕСА С ШЕСТОГО МОДУЛЯ
           #index := 6+#Offset_array_bits;//заполнять функцию будем через индекс чтобы меньше писать
           "rcvDataWeight"(ADDR_DEVICE := #arrayAddressModbus[#index],
                           Ton_changeStep := #Seneca.TON_changeStep.Q,
                           Ton_Start := #Seneca.TON_Start,
                           "Step" := #Seneca.Step,
                           MB_MASTER := #Data_toMB_MASTER);

       12:// КАЛИБРОВКА 0 ДЛЯ ПЯТОГО  МОДУЛЯ

           #index := 5+#Offset_array_bits;//заполнять функцию будем через индекс чтобы меньше писать
           "sndCALIBR&Tara"(ADDR_DEVICE := #arrayAddressModbus[#index],
                        ton_changeStep := #Seneca.TON_changeStep.Q,
                        MB_MASTER := #Data_toMB_MASTER,
                        Ton_Start := #Seneca.TON_Start,
                        Calibrate := #calibrateZero[#index],
                        Buffer := "bufferModBus".Buffer_DataModbusPort1,
                        "Step" := #Seneca.Step,
                        Tara := #taraZero[#index]);

       13:// КАЛИБРОВКА 0 ДЛЯ ШЕСТОГО МОДУЛЯ
           #index := 6+#Offset_array_bits;//заполнять функцию будем через индекс чтобы меньше писать
           "sndCALIBR&Tara"(ADDR_DEVICE := #arrayAddressModbus[#index],
                        ton_changeStep := #Seneca.TON_changeStep.Q,
                        MB_MASTER := #Data_toMB_MASTER,
                        Ton_Start := #Seneca.TON_Start,
                        Calibrate := #calibrateZero[#index],
                        Buffer := "bufferModBus".Buffer_DataModbusPort1,
                        "Step" := #Seneca.Step,
                        Tara := #taraZero[#index]);
   14://отправка аналоговых значений вибрации
       "sndVibration"(ADDR_DEVICE:=40,
                      ton_changeStep:= #Seneca.TON_changeStep.Q,
                      MB_MASTER:=#Data_toMB_MASTER,
                      Ton_Start:=#Seneca.TON_Start,
                      Buffer:="bufferModBus".Buffer_DataModbusPort1,
                      "Step":=#Seneca.Step);
   ELSE
           #Seneca.Step := 1;
   END_CASE;
END_REGION

REGION Network 3: ПРИЕМ ДАННЫХ
   RUNG wire#powerrail
      #MB_MASTER.MB_MASTER(REQ := #Data_toMB_MASTER.REQ, MB_ADDR := #Data_toMB_MASTER.MB_ADDR, MODE := #Data_toMB_MASTER.MODE, DATA_ADDR := #Data_toMB_MASTER.DATA_ADDR, DATA_LEN := #Data_toMB_MASTER.DATA_LEN, DATA_PTR := "bufferModBus".Buffer_DataModbusPort1, DONE => #Data_toMB_MASTER.DONE, BUSY => #Data_toMB_MASTER.BUSY, ERROR => #Data_toMB_MASTER.ERROR, STATUS =>)
   END_RUNG
   // the same network as SCL:
   #MB_MASTER(REQ := #Data_toMB_MASTER.REQ,   // MB_MASTER
              MB_ADDR := #Data_toMB_MASTER.MB_ADDR,
              MODE := #Data_toMB_MASTER.MODE,
              DATA_ADDR := #Data_toMB_MASTER.DATA_ADDR,
              DATA_LEN := #Data_toMB_MASTER.DATA_LEN,
              DATA_PTR := "bufferModBus".Buffer_DataModbusPort1,
              DONE => #Data_toMB_MASTER.DONE,
              BUSY => #Data_toMB_MASTER.BUSY,
              ERROR => #Data_toMB_MASTER.ERROR);
END_REGION

REGION Network 4 (SCL): Авария опроса модуля
   #index := 0;
   CASE #Seneca.Step OF
       2,4:
           #index := 1;
       3,5:
           #index := 2;
       6,8:
           #index := 3;
       7,9:
           #index := 4;
       10,12:
           #index := 5;
       11,13:
           #index := 6;

   END_CASE;
   IF #Data_toMB_MASTER.ERROR THEN
       "hmi".alarmTest.bit[#index] := true;
   ELSIF #Data_toMB_MASTER.DONE THEN
       "hmi".alarmTest.bit[#index] := FALSE;
   END_IF;
END_REGION

REGION Network 5 (SCL)
   IF #Seneca.Step = 2 AND #Data_toMB_MASTER.DONE THEN
       #tmpIndex := 1 + #Offset_array_bits;
       #tmpWeight[#tmpIndex].%W0 := "bufferModBus".Buffer_DataModbusPort1[1];
       #tmpWeight[#tmpIndex].%W1 := "bufferModBus".Buffer_DataModbusPort1[0];
       #currentWeight[#tmpIndex] := DWORD_TO_REAL(#tmpWeight[#tmpIndex]);
       "bufferModBus".Buffer_DataModbusPort1[0] := 0;
       "bufferModBus".Buffer_DataModbusPort1[1] := 0;

   END_IF;

   IF #Seneca.Step = 3 AND #Data_toMB_MASTER.DONE THEN
       #tmpIndex := 2 + #Offset_array_bits;
       #tmpWeight[#tmpIndex].%W0 := "bufferModBus".Buffer_DataModbusPort1[1];
       #tmpWeight[#tmpIndex].%W1 := "bufferModBus".Buffer_DataModbusPort1[0];
       #currentWeight[#tmpIndex] := DWORD_TO_REAL(#tmpWeight[#tmpIndex]);
       "bufferModBus".Buffer_DataModbusPort1[0] := 0;
       "bufferModBus".Buffer_DataModbusPort1[1] := 0;
   END_IF;

   IF #Seneca.Step = 6 AND #Data_toMB_MASTER.DONE THEN
       #tmpIndex := 3 + #Offset_array_bits;
       #tmpWeight[#tmpIndex].%W0 := "bufferModBus".Buffer_DataModbusPort1[1];
       #tmpWeight[#tmpIndex].%W1 := "bufferModBus".Buffer_DataModbusPort1[0];
       #currentWeight[#tmpIndex] := DWORD_TO_REAL(#tmpWeight[#tmpIndex]);
       "bufferModBus".Buffer_DataModbusPort1[0] := 0;
       "bufferModBus".Buffer_DataModbusPort1[1] := 0;
   END_IF;

   IF #Seneca.Step = 7 AND #Data_toMB_MASTER.DONE THEN
       #tmpIndex := 4 + #Offset_array_bits;
       #tmpWeight[#tmpIndex].%W0 := "bufferModBus".Buffer_DataModbusPort1[1];
       #tmpWeight[#tmpIndex].%W1 := "bufferModBus".Buffer_DataModbusPort1[0];
       #currentWeight[#tmpIndex] := DWORD_TO_REAL(#tmpWeight[#tmpIndex]);
       "bufferModBus".Buffer_DataModbusPort1[0] := 0;
       "bufferModBus".Buffer_DataModbusPort1[1] := 0;
   END_IF;

   IF #Seneca.Step = 10 AND #Data_toMB_MASTER.DONE THEN
       #tmpIndex := 5 + #Offset_array_bits;
       #tmpWeight[#tmpIndex].%W0 := "bufferModBus".Buffer_DataModbusPort1[1];
       #tmpWeight[#tmpIndex].%W1 := "bufferModBus".Buffer_DataModbusPort1[0];
       #currentWeight[#tmpIndex] := DWORD_TO_REAL(#tmpWeight[#tmpIndex]);
       "bufferModBus".Buffer_DataModbusPort1[0] := 0;
       "bufferModBus".Buffer_DataModbusPort1[1] := 0;
   END_IF;

   IF #Seneca.Step = 11 AND #Data_toMB_MASTER.DONE THEN
       #tmpIndex := 6 + #Offset_array_bits;
       #tmpWeight[#tmpIndex].%W0 := "bufferModBus".Buffer_DataModbusPort1[1];
       #tmpWeight[#tmpIndex].%W1 := "bufferModBus".Buffer_DataModbusPort1[0];
       #currentWeight[#tmpIndex] := DWORD_TO_REAL(#tmpWeight[#tmpIndex]);
       "bufferModBus".Buffer_DataModbusPort1[0] := 0;
       "bufferModBus".Buffer_DataModbusPort1[1] := 0;
   END_IF;
END_REGION

REGION Network 6: ПОДСЧЕТ ЧИСЛА ОПРОСОВ ЗА 5С
   RUNG wire#powerrail
      Contact( "AlwaysTRUE" )
      I_Contact( "IEC_Timer_TEST_HIGH".Q )
      { S7_Templates := "time_type := Time" } "IEC_Timer_TEST".TON(pt := T#2s, et =>)
      Coil( "pulse_high" )
   END_RUNG
   // the same network as SCL:
   "IEC_Timer_TEST".TON(IN := "AlwaysTRUE" AND NOT "IEC_Timer_TEST_HIGH".Q, PT := T#2s);
   "pulse_high" := "IEC_Timer_TEST".Q;
END_REGION

REGION Network 7
   RUNG wire#powerrail
      Contact( "pulse_high" )
      { S7_Templates := "time_type := Time" } "IEC_Timer_TEST_HIGH".TON(pt := T#5s, et =>)
   END_RUNG
   // the same network as SCL:
   "IEC_Timer_TEST_HIGH".TON(IN := "pulse_high", PT := T#5s);
END_REGION

REGION Network 8
   RUNG wire#powerrail
      Contact( #MB_MASTER.DONE )
      P_Trig( "Tag_1" )
      { S7_Templates := "value_type := Int" } "IEC_Counter_0_DB".CTU(r := wire#w1, pv := 32765, cv =>)
   END_RUNG
   RUNG wire#powerrail
      I_Contact( "pulse_high" )
   END_RUNG wire#w1
   // the same network as SCL:
   #_w1 := #MB_MASTER.DONE AND NOT "Tag_1";   // rising edge
   "Tag_1" := #MB_MASTER.DONE;
   "IEC_Counter_0_DB".CTU(CU := #_w1, R := NOT "pulse_high", PV := 32765);
END_REGION
END_FUNCTION_BLOCK

FUNCTION_BLOCK "modbus_SenecaConnectPort2"   // FB14, LAD
{ S7_Optimized_Access := 'TRUE' }
VERSION : 0.1
// stored: AutoNumber false, IsIECCheckEnabled false, IsRetainMemResEnabled false, MemoryReserve 100, SetENOAutomatically false, UDAEnableTagReadback false
   VAR_INPUT
      port : PORT;   // порт для подключения
      arrayAddressModbus : Array[0..12] of UInt;
      Offset_array_bits : SInt;
   END_VAR
   VAR_IN_OUT
      calibrateZero : Array[0..12] of Bool;
      taraZero : Array[0..12] of Bool;
      currentWeight : Array[0..12] of Real;
   END_VAR
   VAR
      MB_COMM_LOAD : MB_COMM_LOAD;
      MB_MASTER : MB_MASTER;
      Data_toMB_MASTER : Struct
         REQ : Bool;
         MB_ADDR : UInt;
         MODE : USInt;
         DATA_ADDR : UDInt;
         DATA_LEN : UInt;
         DONE : Bool;
         BUSY : Bool;
         ERROR : Bool;
      END_STRUCT;
      Seneca : Struct
         TON_changeStep : TON_TIME;
         TON_Start { S7_SetPoint := 'True'} : Bool;
         "Step" : SInt;
      END_STRUCT;
      tmpWeight : Array[0..12] of DWord;
      restartPort : Bool;   // перезагрузка Modbus
   END_VAR
   VAR_TEMP
      index : DInt;
      tmpIndex : DInt;
   END_VAR
   // MB_COMM_LOAD.RETRIES := 1;
BEGIN

REGION Network 1: ИНИЦИАЛИЗИРУЕМ ПОРТ
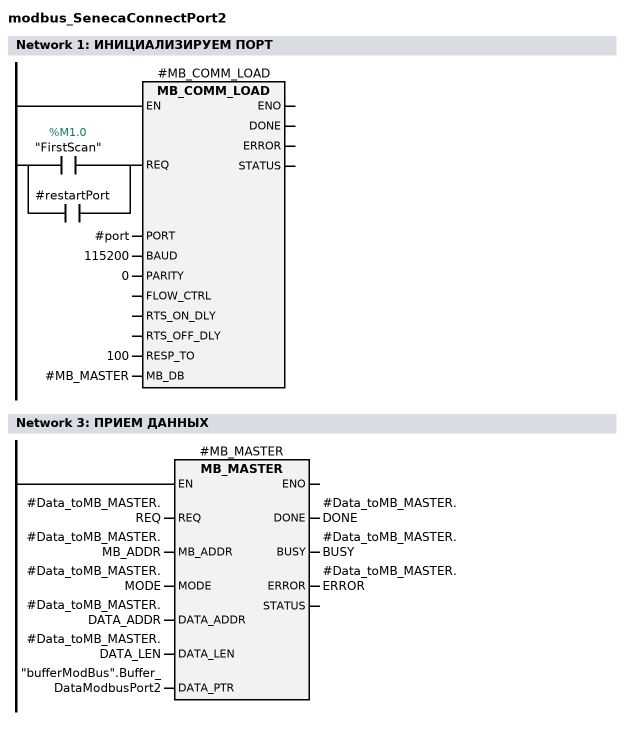
   RUNG wire#powerrail
      #MB_COMM_LOAD.MB_COMM_LOAD(REQ := wire#w1, PORT := #port, BAUD := 115200, PARITY := 0, FLOW_CTRL :=, RTS_ON_DLY :=, RTS_OFF_DLY :=, RESP_TO := 100, MB_DB := #MB_MASTER, DONE =>, ERROR =>, STATUS =>)
   END_RUNG
   RUNG wire#powerrail
      Contact( "FirstScan" )
   END_RUNG wire#w1
   RUNG wire#powerrail
      Contact( #restartPort )
   END_RUNG wire#w1
   // the same network as SCL:
   #MB_COMM_LOAD(REQ := "FirstScan" OR #restartPort,   // MB_COMM_LOAD
                 PORT := #port,
                 BAUD := 115200,
                 PARITY := 0,
                 RESP_TO := 100,
                 MB_DB := #MB_MASTER);
END_REGION

REGION Network 2 (SCL): ОБМЕН
   #Seneca.TON_changeStep(IN :=#Seneca.TON_Start,
                          PT := t#50ms);

   CASE #Seneca.Step OF

       1:
           #Seneca.Step := #Seneca.Step + 1;

       2: //ЧИТАЕМ ЗНАЧЕНИЕ ВЕСА С ПЕРВОГО МОДУЛЯ

           #index := 1+#Offset_array_bits;//заполнять функцию будем через индекс чтобы меньше писать
           "rcvDataWeight"(ADDR_DEVICE := #arrayAddressModbus[#index],
                           Ton_changeStep:=#Seneca.TON_changeStep.Q,
                           Ton_Start:=#Seneca.TON_Start,
                           "Step":=#Seneca.Step,
                           MB_MASTER:=#Data_toMB_MASTER);

       3://ЧИТАЕМ ЗНАЧЕНИЕ ВЕСА СО ВТОРОГО МОДУЛЯ
           #index := 2+#Offset_array_bits;//заполнять функцию будем через индекс чтобы меньше писать
           "rcvDataWeight"(ADDR_DEVICE := #arrayAddressModbus[#index],
                           Ton_changeStep:=#Seneca.TON_changeStep.Q,
                           Ton_Start:=#Seneca.TON_Start,
                           "Step":=#Seneca.Step,
                           MB_MASTER:=#Data_toMB_MASTER);

       4: // КАЛИБРОВКА 0 ДЛЯ ПЕРВОГО МОДУЛЯ и ТАРИРОВАНИЕ
           #index := 1+#Offset_array_bits;//заполнять функцию будем через индекс чтобы меньше писать
           "sndCALIBR&Tara"(ADDR_DEVICE := #arrayAddressModbus[#index],
                            ton_changeStep:=#Seneca.TON_changeStep.Q,
                        MB_MASTER:=#Data_toMB_MASTER,
                        Ton_Start:=#Seneca.TON_Start,
                        Calibrate:=#calibrateZero[#index],
                        Buffer:="bufferModBus".Buffer_DataModbusPort2,
                        "Step":=#Seneca.Step,
                        Tara:=#taraZero[#index]);

       5:// КАЛИБРОВКА 0 ДЛЯ ВТОРОГО МОДУЛЯ и ТАРИРОВАНИЕ
           #index := 2+#Offset_array_bits;//заполнять функцию будем через индекс чтобы меньше писать
           "sndCALIBR&Tara"(ADDR_DEVICE := #arrayAddressModbus[#index],
                            ton_changeStep := #Seneca.TON_changeStep.Q,
                        MB_MASTER := #Data_toMB_MASTER,
                        Ton_Start := #Seneca.TON_Start,
                        Calibrate := #calibrateZero[#index],
                        Buffer := "bufferModBus".Buffer_DataModbusPort2,
                        "Step" := #Seneca.Step,
                        Tara := #taraZero[#index]);

           //////////////////////////////////////////////////////////////////////////////////
           //////////////////////////////////////////////////////////////////////////////////
           //////////////////////////////////////////////////////////////////////////////////
           //////////////////////////////////////////////////////////////////////////////////
       6: //ЧИТАЕМ ЗНАЧЕНИЕ ВЕСА С ТРЕТЬЕГО МОДУЛЯ

           #index := 3+#Offset_array_bits;//заполнять функцию будем через индекс чтобы меньше писать
           "rcvDataWeight"(ADDR_DEVICE := #arrayAddressModbus[#index],
                           Ton_changeStep := #Seneca.TON_changeStep.Q,
                           Ton_Start := #Seneca.TON_Start,
                           "Step" := #Seneca.Step,
                           MB_MASTER := #Data_toMB_MASTER);

       7://ЧИТАЕМ ЗНАЧЕНИЕ ВЕСА С ЧЕТВЕРТОГО МОДУЛЯ
           #index := 4+#Offset_array_bits;//заполнять функцию будем через индекс чтобы меньше писать
           "rcvDataWeight"(ADDR_DEVICE := #arrayAddressModbus[#index],
                           Ton_changeStep := #Seneca.TON_changeStep.Q,
                           Ton_Start := #Seneca.TON_Start,
                           "Step" := #Seneca.Step,
                           MB_MASTER := #Data_toMB_MASTER);

       8:// КАЛИБРОВКА 0 ДЛЯ ТРЕТЬЕГО  МОДУЛЯ

           #index := 3+#Offset_array_bits;//заполнять функцию будем через индекс чтобы меньше писать
           "sndCALIBR&Tara"(ADDR_DEVICE := #arrayAddressModbus[#index],
                            ton_changeStep := #Seneca.TON_changeStep.Q,
                        MB_MASTER := #Data_toMB_MASTER,
                        Ton_Start := #Seneca.TON_Start,
                        Calibrate := #calibrateZero[#index],
                        Buffer := "bufferModBus".Buffer_DataModbusPort2,
                        "Step" := #Seneca.Step,
                        Tara := #taraZero[#index]);

       9://КАЛИБРОВКА 0 ДЛЯ ЧЕТВЕРТОГО МОДУЛЯ

           #index := 4+#Offset_array_bits;//заполнять функцию будем через индекс чтобы меньше писать
           "sndCALIBR&Tara"(ADDR_DEVICE := #arrayAddressModbus[#index],
                            ton_changeStep := #Seneca.TON_changeStep.Q,
                        MB_MASTER := #Data_toMB_MASTER,
                        Ton_Start := #Seneca.TON_Start,
                        Calibrate := #calibrateZero[#index],
                        Buffer := "bufferModBus".Buffer_DataModbusPort2,
                        "Step" := #Seneca.Step,
                        Tara := #taraZero[#index]);

           /////////////////////////////////////////////////////////////////////////////////
           ////////////////////////////////////////////////////////////////////////////////
           ////////////////////////////////////////////////////////////////////////////////
           ////////////////////////////////////////////////////////////////////////////////
       10: //ЧИТАЕМ ЗНАЧЕНИЕ ВЕСА С ПЯТОГО МОДУЛЯ
           #index := 5+#Offset_array_bits;//заполнять функцию будем через индекс чтобы меньше писать
           "rcvDataWeight"(ADDR_DEVICE := #arrayAddressModbus[#index],
                           Ton_changeStep := #Seneca.TON_changeStep.Q,
                           Ton_Start := #Seneca.TON_Start,
                           "Step" := #Seneca.Step,
                           MB_MASTER := #Data_toMB_MASTER);

       11://ЧИТАЕМ ЗНАЧЕНИЕ ВЕСА С ШЕСТОГО МОДУЛЯ
           #index := 6+#Offset_array_bits;//заполнять функцию будем через индекс чтобы меньше писать
           "rcvDataWeight"(ADDR_DEVICE := #arrayAddressModbus[#index],
                           Ton_changeStep := #Seneca.TON_changeStep.Q,
                           Ton_Start := #Seneca.TON_Start,
                           "Step" := #Seneca.Step,
                           MB_MASTER := #Data_toMB_MASTER);

       12:// КАЛИБРОВКА 0 ДЛЯ ПЯТОГО  МОДУЛЯ

           #index := 5+#Offset_array_bits;//заполнять функцию будем через индекс чтобы меньше писать
           "sndCALIBR&Tara"(ADDR_DEVICE := #arrayAddressModbus[#index],
                        ton_changeStep := #Seneca.TON_changeStep.Q,
                        MB_MASTER := #Data_toMB_MASTER,
                        Ton_Start := #Seneca.TON_Start,
                        Calibrate := #calibrateZero[#index],
                        Buffer := "bufferModBus".Buffer_DataModbusPort2,
                        "Step" := #Seneca.Step,
                        Tara := #taraZero[#index]);

       13:// КАЛИБРОВКА 0 ДЛЯ ШЕСТОГО МОДУЛЯ
           #index := 6+#Offset_array_bits;//заполнять функцию будем через индекс чтобы меньше писать
           "sndCALIBR&Tara"(ADDR_DEVICE := #arrayAddressModbus[#index],
                            ton_changeStep := #Seneca.TON_changeStep.Q,
                        MB_MASTER := #Data_toMB_MASTER,
                        Ton_Start := #Seneca.TON_Start,
                        Calibrate := #calibrateZero[#index],
                        Buffer := "bufferModBus".Buffer_DataModbusPort2,
                        "Step" := #Seneca.Step,
                        Tara := #taraZero[#index]);
       ELSE
           #Seneca.Step := 1;
   END_CASE;
END_REGION

REGION Network 3: ПРИЕМ ДАННЫХ
   RUNG wire#powerrail
      #MB_MASTER.MB_MASTER(REQ := #Data_toMB_MASTER.REQ, MB_ADDR := #Data_toMB_MASTER.MB_ADDR, MODE := #Data_toMB_MASTER.MODE, DATA_ADDR := #Data_toMB_MASTER.DATA_ADDR, DATA_LEN := #Data_toMB_MASTER.DATA_LEN, DATA_PTR := "bufferModBus".Buffer_DataModbusPort2, DONE => #Data_toMB_MASTER.DONE, BUSY => #Data_toMB_MASTER.BUSY, ERROR => #Data_toMB_MASTER.ERROR, STATUS =>)
   END_RUNG
   // the same network as SCL:
   #MB_MASTER(REQ := #Data_toMB_MASTER.REQ,   // MB_MASTER
              MB_ADDR := #Data_toMB_MASTER.MB_ADDR,
              MODE := #Data_toMB_MASTER.MODE,
              DATA_ADDR := #Data_toMB_MASTER.DATA_ADDR,
              DATA_LEN := #Data_toMB_MASTER.DATA_LEN,
              DATA_PTR := "bufferModBus".Buffer_DataModbusPort2,
              DONE => #Data_toMB_MASTER.DONE,
              BUSY => #Data_toMB_MASTER.BUSY,
              ERROR => #Data_toMB_MASTER.ERROR);
END_REGION

REGION Network 4 (SCL): Авария опроса модуля
   #index := 0;
   CASE #Seneca.Step OF
       2,4:
           #index := 7;
       3,5:
           #index := 8;
       6,8:
           #index := 9;
       7,9:
           #index := 10;
       10,12:
           #index := 11;
       11,13:
           #index := 12;

   END_CASE;
   IF #Data_toMB_MASTER.ERROR THEN
       "hmi".alarmTest.bit[#index] := true;
   ELSIF #Data_toMB_MASTER.DONE THEN
       "hmi".alarmTest.bit[#index] := FALSE;
   END_IF;
END_REGION

REGION Network 5 (SCL)
   IF #Seneca.Step = 2 AND #Data_toMB_MASTER.DONE THEN
       #tmpIndex := 1 + #Offset_array_bits;
       #tmpWeight[#tmpIndex].%W0 := "bufferModBus".Buffer_DataModbusPort2[1];
       #tmpWeight[#tmpIndex].%W1 := "bufferModBus".Buffer_DataModbusPort2[0];
       #currentWeight[#tmpIndex] := DWORD_TO_REAL(#tmpWeight[#tmpIndex]);
       "bufferModBus".Buffer_DataModbusPort2[0] := 0;
       "bufferModBus".Buffer_DataModbusPort2[1] := 0;

   END_IF;

   IF #Seneca.Step = 3 AND #Data_toMB_MASTER.DONE THEN
       #tmpIndex := 2 + #Offset_array_bits;
       #tmpWeight[#tmpIndex].%W0 := "bufferModBus".Buffer_DataModbusPort2[1];
       #tmpWeight[#tmpIndex].%W1 := "bufferModBus".Buffer_DataModbusPort2[0];
       #currentWeight[#tmpIndex] := DWORD_TO_REAL(#tmpWeight[#tmpIndex]);
       "bufferModBus".Buffer_DataModbusPort2[0] := 0;
       "bufferModBus".Buffer_DataModbusPort2[1] := 0;
   END_IF;

   IF #Seneca.Step = 6 AND #Data_toMB_MASTER.DONE THEN
       #tmpIndex := 3 + #Offset_array_bits;
       #tmpWeight[#tmpIndex].%W0 := "bufferModBus".Buffer_DataModbusPort2[1];
       #tmpWeight[#tmpIndex].%W1 := "bufferModBus".Buffer_DataModbusPort2[0];
       #currentWeight[#tmpIndex] := DWORD_TO_REAL(#tmpWeight[#tmpIndex]);
       "bufferModBus".Buffer_DataModbusPort2[0] := 0;
       "bufferModBus".Buffer_DataModbusPort2[1] := 0;
   END_IF;

   IF #Seneca.Step = 7 AND #Data_toMB_MASTER.DONE THEN
       #tmpIndex := 4 + #Offset_array_bits;
       #tmpWeight[#tmpIndex].%W0 := "bufferModBus".Buffer_DataModbusPort2[1];
       #tmpWeight[#tmpIndex].%W1 := "bufferModBus".Buffer_DataModbusPort2[0];
       #currentWeight[#tmpIndex] := DWORD_TO_REAL(#tmpWeight[#tmpIndex]);
       "bufferModBus".Buffer_DataModbusPort2[0] := 0;
       "bufferModBus".Buffer_DataModbusPort2[1] := 0;
   END_IF;

   IF #Seneca.Step = 10 AND #Data_toMB_MASTER.DONE THEN
       #tmpIndex := 5 + #Offset_array_bits;
       #tmpWeight[#tmpIndex].%W0 := "bufferModBus".Buffer_DataModbusPort2[1];
       #tmpWeight[#tmpIndex].%W1 := "bufferModBus".Buffer_DataModbusPort2[0];
       #currentWeight[#tmpIndex] := DWORD_TO_REAL(#tmpWeight[#tmpIndex]);
       "bufferModBus".Buffer_DataModbusPort2[0] := 0;
       "bufferModBus".Buffer_DataModbusPort2[1] := 0;
   END_IF;

   IF #Seneca.Step = 11 AND #Data_toMB_MASTER.DONE THEN
       #tmpIndex := 6 + #Offset_array_bits;
       #tmpWeight[#tmpIndex].%W0 := "bufferModBus".Buffer_DataModbusPort2[1];
       #tmpWeight[#tmpIndex].%W1 := "bufferModBus".Buffer_DataModbusPort2[0];
       #currentWeight[#tmpIndex] := DWORD_TO_REAL(#tmpWeight[#tmpIndex]);
       "bufferModBus".Buffer_DataModbusPort2[0] := 0;
       "bufferModBus".Buffer_DataModbusPort2[1] := 0;
   END_IF;
END_REGION
END_FUNCTION_BLOCK

FUNCTION "IOtoDB" : Void   // FC1, LAD
{ S7_Optimized_Access := 'TRUE' }
VERSION : 0.1
// stored: AutoNumber false, IsIECCheckEnabled false, SetENOAutomatically false, UDAEnableTagReadback false
BEGIN

REGION Network 1: Передаем входа
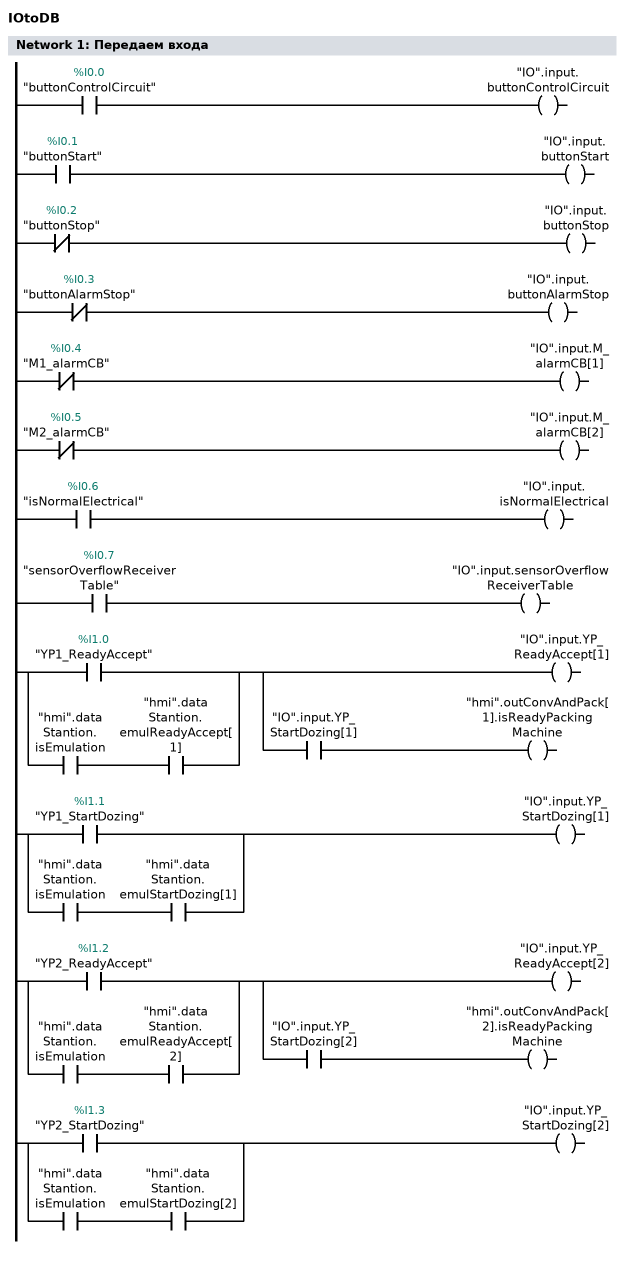
   RUNG wire#powerrail
      Contact( "buttonControlCircuit" )
      Coil( "IO".input.buttonControlCircuit )
   END_RUNG
   RUNG wire#powerrail
      Contact( "buttonStart" )
      Coil( "IO".input.buttonStart )
   END_RUNG
   RUNG wire#powerrail
      I_Contact( "buttonStop" )
      Coil( "IO".input.buttonStop )
   END_RUNG
   RUNG wire#powerrail
      I_Contact( "buttonAlarmStop" )
      Coil( "IO".input.buttonAlarmStop )
   END_RUNG
   RUNG wire#powerrail
      I_Contact( "M1_alarmCB" )
      Coil( "IO".input.M_alarmCB[1] )
   END_RUNG
   RUNG wire#powerrail
      I_Contact( "M2_alarmCB" )
      Coil( "IO".input.M_alarmCB[2] )
   END_RUNG
   RUNG wire#powerrail
      Contact( "isNormalElectrical" )
      Coil( "IO".input.isNormalElectrical )
   END_RUNG
   RUNG wire#powerrail
      Contact( "sensorOverflowReceiverTable" )
      Coil( "IO".input.sensorOverflowReceiverTable )
   END_RUNG
   RUNG wire#powerrail
      Contact( "YP1_ReadyAccept" )
      wire#w1
      Coil( "IO".input.YP_ReadyAccept[1] )
   END_RUNG
   RUNG wire#powerrail
      Contact( "hmi".dataStantion.isEmulation )
      Contact( "hmi".dataStantion.emulReadyAccept[1] )
   END_RUNG wire#w1
   RUNG wire#w1
      Contact( "IO".input.YP_StartDozing[1] )
      Coil( "hmi".outConvAndPack[1].isReadyPackingMachine )
   END_RUNG
   RUNG wire#powerrail
      Contact( "YP1_StartDozing" )
      wire#w2
      Coil( "IO".input.YP_StartDozing[1] )
   END_RUNG
   RUNG wire#powerrail
      Contact( "hmi".dataStantion.isEmulation )
      Contact( "hmi".dataStantion.emulStartDozing[1] )
   END_RUNG wire#w2
   RUNG wire#powerrail
      Contact( "YP2_ReadyAccept" )
      wire#w3
      Coil( "IO".input.YP_ReadyAccept[2] )
   END_RUNG
   RUNG wire#powerrail
      Contact( "hmi".dataStantion.isEmulation )
      Contact( "hmi".dataStantion.emulReadyAccept[2] )
   END_RUNG wire#w3
   RUNG wire#w3
      Contact( "IO".input.YP_StartDozing[2] )
      Coil( "hmi".outConvAndPack[2].isReadyPackingMachine )
   END_RUNG
   RUNG wire#powerrail
      Contact( "YP2_StartDozing" )
      wire#w4
      Coil( "IO".input.YP_StartDozing[2] )
   END_RUNG
   RUNG wire#powerrail
      Contact( "hmi".dataStantion.isEmulation )
      Contact( "hmi".dataStantion.emulStartDozing[2] )
   END_RUNG wire#w4
   // the same network as SCL:
   "IO".input.buttonControlCircuit := "buttonControlCircuit";
   "IO".input.buttonStart := "buttonStart";
   "IO".input.buttonStop := NOT "buttonStop";
   "IO".input.buttonAlarmStop := NOT "buttonAlarmStop";
   "IO".input.M_alarmCB[1] := NOT "M1_alarmCB";
   "IO".input.M_alarmCB[2] := NOT "M2_alarmCB";
   "IO".input.isNormalElectrical := "isNormalElectrical";
   "IO".input.sensorOverflowReceiverTable := "sensorOverflowReceiverTable";
   "IO".input.YP_ReadyAccept[1] := "YP1_ReadyAccept" OR ("hmi".dataStantion.isEmulation AND "hmi".dataStantion.emulReadyAccept[1]);
   "hmi".outConvAndPack[1].isReadyPackingMachine := ("YP1_ReadyAccept" OR ("hmi".dataStantion.isEmulation AND "hmi".dataStantion.emulReadyAccept[1])) AND "IO".input.YP_StartDozing[1];
   "IO".input.YP_StartDozing[1] := "YP1_StartDozing" OR ("hmi".dataStantion.isEmulation AND "hmi".dataStantion.emulStartDozing[1]);
   "IO".input.YP_ReadyAccept[2] := "YP2_ReadyAccept" OR ("hmi".dataStantion.isEmulation AND "hmi".dataStantion.emulReadyAccept[2]);
   "hmi".outConvAndPack[2].isReadyPackingMachine := ("YP2_ReadyAccept" OR ("hmi".dataStantion.isEmulation AND "hmi".dataStantion.emulReadyAccept[2])) AND "IO".input.YP_StartDozing[2];
   "IO".input.YP_StartDozing[2] := "YP2_StartDozing" OR ("hmi".dataStantion.isEmulation AND "hmi".dataStantion.emulStartDozing[2]);
END_REGION
END_FUNCTION

FUNCTION "preWorkBlock" : Void   // FC9, LAD
TITLE = Блок предработы
{ S7_Optimized_Access := 'TRUE' }
VERSION : 0.1
// Блок в котором организована работа цепей управления, аварийного останова и режимов работы
// stored: AutoNumber false, IsIECCheckEnabled false, SetENOAutomatically false, UDAEnableTagReadback false
BEGIN

REGION Network 1: удержание кнопки включение цепей управления
   // если аварийная кнопка не нажата то держим 2 секунды и цепи управления включаются
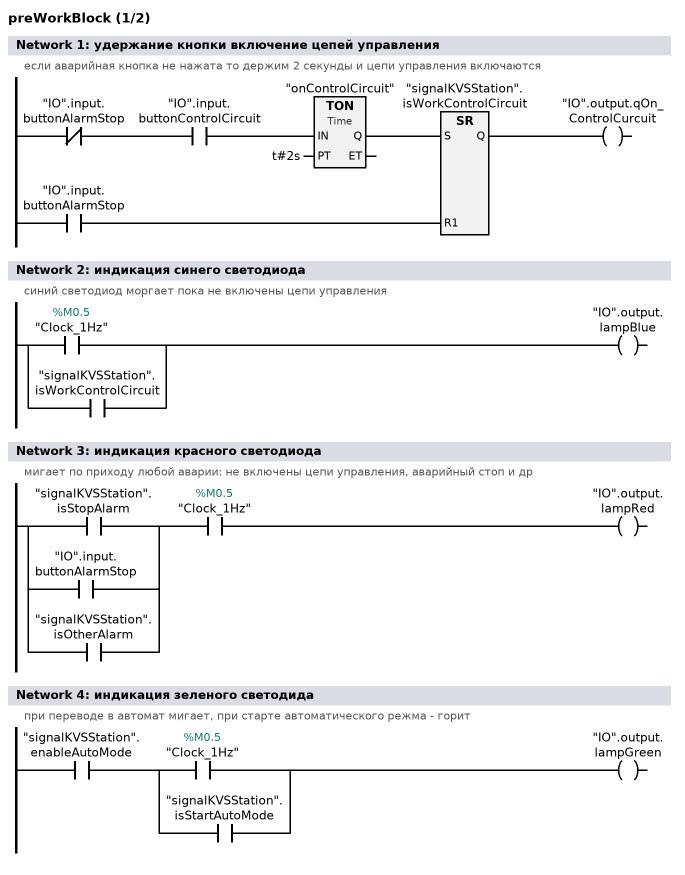
   RUNG wire#powerrail
      I_Contact( "IO".input.buttonAlarmStop )
      Contact( "IO".input.buttonControlCircuit )
      { S7_Templates := "time_type := Time" } "onControlCircuit".TON(pt := t#2s, et =>)
      S_SR(operand := "signalKVSStation".isWorkControlCircuit, r1 := wire#w1)
      Coil( "IO".output.qOn_ControlCurcuit )
   END_RUNG
   RUNG wire#powerrail
      Contact( "IO".input.buttonAlarmStop )
   END_RUNG wire#w1
   // the same network as SCL:
   "onControlCircuit".TON(IN := NOT "IO".input.buttonAlarmStop AND "IO".input.buttonControlCircuit, PT := t#2s);
   IF "onControlCircuit".Q THEN
       "signalKVSStation".isWorkControlCircuit := TRUE;   // SR flip-flop
   END_IF;
   IF "IO".input.buttonAlarmStop THEN "signalKVSStation".isWorkControlCircuit := FALSE; END_IF;
   "IO".output.qOn_ControlCurcuit := "signalKVSStation".isWorkControlCircuit;
END_REGION

REGION Network 2: индикация синего светодиода
   // синий светодиод моргает пока не включены цепи управления
   RUNG wire#powerrail
      Contact( "Clock_1Hz" )
      wire#w1
      Coil( "IO".output.lampBlue )
   END_RUNG
   RUNG wire#powerrail
      Contact( "signalKVSStation".isWorkControlCircuit )
   END_RUNG wire#w1
   // the same network as SCL:
   "IO".output.lampBlue := "Clock_1Hz" OR "signalKVSStation".isWorkControlCircuit;
END_REGION

REGION Network 3: индикация красного светодиода
   // мигает по приходу любой аварии: не включены цепи управления, аварийный стоп и др
   RUNG wire#powerrail
      Contact( "signalKVSStation".isStopAlarm )
      wire#w1
      Contact( "Clock_1Hz" )
      Coil( "IO".output.lampRed )
   END_RUNG
   RUNG wire#powerrail
      Contact( "IO".input.buttonAlarmStop )
   END_RUNG wire#w1
   RUNG wire#powerrail
      Contact( "signalKVSStation".isOtherAlarm )
   END_RUNG wire#w1
   // the same network as SCL:
   "IO".output.lampRed := ("signalKVSStation".isStopAlarm OR "IO".input.buttonAlarmStop OR "signalKVSStation".isOtherAlarm) AND "Clock_1Hz";
END_REGION

REGION Network 4: индикация зеленого светодида
   // при переводе в автомат мигает, при старте автоматического режма - горит
   RUNG wire#powerrail
      Contact( "signalKVSStation".enableAutoMode )
      wire#w1
      Contact( "Clock_1Hz" )
      wire#w2
      Coil( "IO".output.lampGreen )
   END_RUNG
   RUNG wire#w1
      Contact( "signalKVSStation".isStartAutoMode )
   END_RUNG wire#w2
   // the same network as SCL:
   "IO".output.lampGreen := "signalKVSStation".enableAutoMode AND ("Clock_1Hz" OR "signalKVSStation".isStartAutoMode);
END_REGION

REGION Network 5: разрешение на перевод в автоматический режим
   // при отсутствии аварий и нажатии кнопки автотоматического режима на панели. Данный сигнал используется как обратная связь по автоматическому и ручному режиму
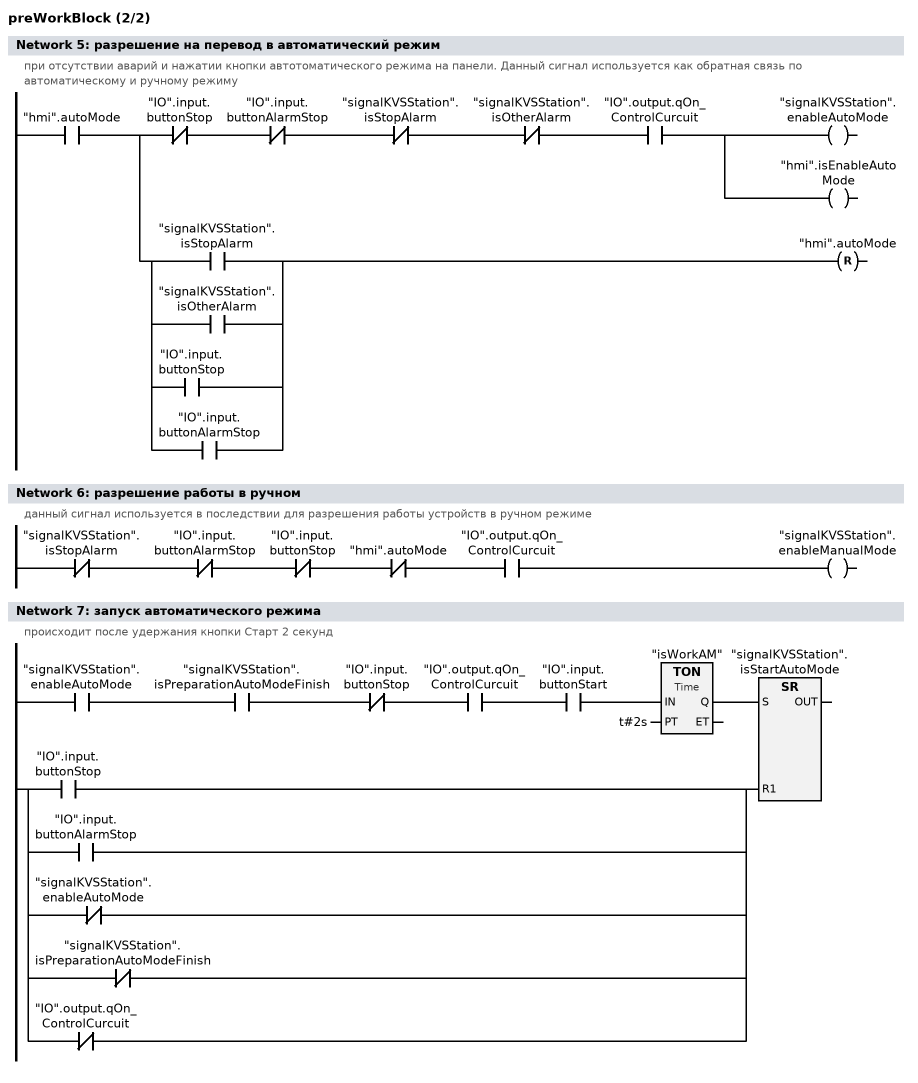
   RUNG wire#powerrail
      Contact( "hmi".autoMode )
      wire#w1
      I_Contact( "IO".input.buttonStop )
      I_Contact( "IO".input.buttonAlarmStop )
      I_Contact( "signalKVSStation".isStopAlarm )
      I_Contact( "signalKVSStation".isOtherAlarm )
      Contact( "IO".output.qOn_ControlCurcuit )
      wire#w2
      Coil( "signalKVSStation".enableAutoMode )
   END_RUNG
   RUNG wire#w2
      Coil( "hmi".isEnableAutoMode )
   END_RUNG
   RUNG wire#w1
      Contact( "signalKVSStation".isStopAlarm )
      wire#w3
      R_Coil( "hmi".autoMode )
   END_RUNG
   RUNG wire#w1
      Contact( "signalKVSStation".isOtherAlarm )
   END_RUNG wire#w3
   RUNG wire#w1
      Contact( "IO".input.buttonStop )
   END_RUNG wire#w3
   RUNG wire#w1
      Contact( "IO".input.buttonAlarmStop )
   END_RUNG wire#w3
   // the same network as SCL:
   "signalKVSStation".enableAutoMode := "hmi".autoMode AND NOT "IO".input.buttonStop AND NOT "IO".input.buttonAlarmStop AND NOT "signalKVSStation".isStopAlarm AND NOT "signalKVSStation".isOtherAlarm AND "IO".output.qOn_ControlCurcuit;
   "hmi".isEnableAutoMode := "signalKVSStation".enableAutoMode;
   IF "hmi".autoMode AND ("signalKVSStation".isStopAlarm OR "signalKVSStation".isOtherAlarm OR "IO".input.buttonStop OR "IO".input.buttonAlarmStop) THEN
       "hmi".autoMode := FALSE;
   END_IF;
END_REGION

REGION Network 6: разрешение работы в ручном
   // данный сигнал используется в последствии для разрешения работы устройств в ручном режиме
   RUNG wire#powerrail
      I_Contact( "signalKVSStation".isStopAlarm )
      I_Contact( "IO".input.buttonAlarmStop )
      I_Contact( "IO".input.buttonStop )
      I_Contact( "hmi".autoMode )
      Contact( "IO".output.qOn_ControlCurcuit )
      Coil( "signalKVSStation".enableManualMode )
   END_RUNG
   // the same network as SCL:
   "signalKVSStation".enableManualMode := NOT "signalKVSStation".isStopAlarm AND NOT "IO".input.buttonAlarmStop AND NOT "IO".input.buttonStop AND NOT "hmi".autoMode AND "IO".output.qOn_ControlCurcuit;
END_REGION

REGION Network 7: запуск автоматического режима
   // происходит после удержания кнопки Старт 2 секунд
   RUNG wire#powerrail
      Contact( "signalKVSStation".enableAutoMode )
      Contact( "signalKVSStation".isPreparationAutoModeFinish )
      I_Contact( "IO".input.buttonStop )
      Contact( "IO".output.qOn_ControlCurcuit )
      Contact( "IO".input.buttonStart )
      { S7_Templates := "time_type := Time" } "isWorkAM".TON(pt := t#2s, et =>)
      S_SR(operand := "signalKVSStation".isStartAutoMode, r1 := wire#w1)
   END_RUNG
   RUNG wire#powerrail
      Contact( "IO".input.buttonStop )
   END_RUNG wire#w1
   RUNG wire#powerrail
      Contact( "IO".input.buttonAlarmStop )
   END_RUNG wire#w1
   RUNG wire#powerrail
      I_Contact( "signalKVSStation".enableAutoMode )
   END_RUNG wire#w1
   RUNG wire#powerrail
      I_Contact( "signalKVSStation".isPreparationAutoModeFinish )
   END_RUNG wire#w1
   RUNG wire#powerrail
      I_Contact( "IO".output.qOn_ControlCurcuit )
   END_RUNG wire#w1
   // the same network as SCL:
   "isWorkAM".TON(IN := "signalKVSStation".enableAutoMode AND "signalKVSStation".isPreparationAutoModeFinish AND NOT "IO".input.buttonStop AND "IO".output.qOn_ControlCurcuit AND "IO".input.buttonStart,
                  PT := t#2s);
   IF "isWorkAM".Q THEN
       "signalKVSStation".isStartAutoMode := TRUE;   // SR flip-flop
   END_IF;
   IF "IO".input.buttonStop OR "IO".input.buttonAlarmStop OR NOT "signalKVSStation".enableAutoMode OR NOT "signalKVSStation".isPreparationAutoModeFinish OR NOT "IO".output.qOn_ControlCurcuit THEN
       "signalKVSStation".isStartAutoMode := FALSE;
   END_IF;
END_REGION
END_FUNCTION

FUNCTION_BLOCK "ManualMode"   // FB10, LAD
{ S7_Optimized_Access := 'TRUE' }
VERSION : 0.1
// stored: AutoNumber false, IsIECCheckEnabled false, IsRetainMemResEnabled false, MemoryReserve 100, SetENOAutomatically false, UDAEnableTagReadback false
   VAR
      Bunker_Left : Array[0..12] of "controlValve";
      Bunker_Right : Array[0..12] of "controlValve";
      Door : Array[0..12] of "controlValve";
      flipper : "controlValve";
      runAll : Struct
         vibroLot : Bool;
      END_STRUCT;
      stopAlarm : Bool;   // Стоп для блоков управления задвижками
   END_VAR
   VAR_TEMP
      i : DInt;
   END_VAR
BEGIN

REGION Network 1: формирование AlarmStop
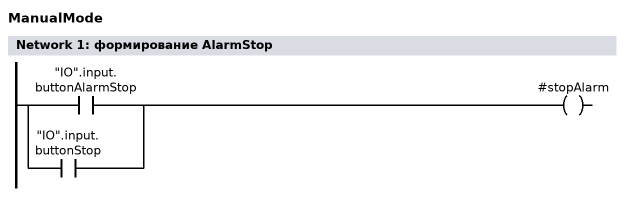
   RUNG wire#powerrail
      Contact( "IO".input.buttonAlarmStop )
      wire#w1
      Coil( #stopAlarm )
   END_RUNG
   RUNG wire#powerrail
      Contact( "IO".input.buttonStop )
   END_RUNG wire#w1
   // the same network as SCL:
   #stopAlarm := "IO".input.buttonAlarmStop OR "IO".input.buttonStop;
END_REGION

REGION Network 2 (SCL): ручное управление
   #i := 0;
   FOR #i := 1 TO 12 DO
       //если имеется разрешение на включение механизмов в ручном режиме
       IF "signalKVSStation".enableManualMode THEN
           //Bunker_left
           #Bunker_Left[#i](openQ => "signalKVSStation".qManualMode.Bunker_leftOpen[#i],
                            closeQ => "signalKVSStation".qManualMode.Bunker_leftClose[#i],
                            open := "hmi".weightLine[#i].manOpenLeftValveWeightPocket,
                            close := "hmi".weightLine[#i].manCloseLeftValveWeightPocket,
                            "time_open/close" := t#250ms,
                            stopAlarm := #stopAlarm);


           //Bunker_right
           #Bunker_Right[#i](openQ => "signalKVSStation".qManualMode.Bunker_rightOpen[#i],
                             closeQ => "signalKVSStation".qManualMode.Bunker_rightClose[#i],
                             open := "hmi".weightLine[#i].manOpenRightValveWeightPocket,
                             close := "hmi".weightLine[#i].manCloseRightValveWieghtPocket,
                             "time_open/close" := t#250ms,
                             stopAlarm := #stopAlarm);

           //Door
           #Door[#i](openQ => "signalKVSStation".qManualMode.Door_open[#i],
                     closeQ => "signalKVSStation".qManualMode.Door_close[#i],
                     open := "hmi".weightLine[#i].manOpenValveAfterVibroLot,
                     close := "hmi".weightLine[#i].manCloseValveAfterVibroLot,
                     "time_open/close" := t#250ms,
                     stopAlarm := #stopAlarm);

           //vibroLot
           IF "hmi".weightLine[#i].manVibroLotStart THEN
               "signalKVSStation".qManualMode.vibroLot[#i] := true;
           ELSE
               "signalKVSStation".qManualMode.vibroLot[#i] := false;
           END_IF;

           //теперь все что на два цикла
           IF #i = 1 OR #i = 2 THEN

               //Conv_FRV //Conv_REV
               IF "hmi".outConvAndPack[#i].manStartOutConv THEN
                   IF "hmi".outConvAndPack[#i].manIsUpConv THEN
                       "signalKVSStation".qManualMode.Conv_FRV[#i] := true;
                       "signalKVSStation".qManualMode.Conv_REV[#i] := false;
                   ELSE
                       "signalKVSStation".qManualMode.Conv_REV[#i] := true;
                       "signalKVSStation".qManualMode.Conv_FRV[#i] := false;
                   END_IF;
               ELSE
                   "signalKVSStation".qManualMode.Conv_REV[#i] := false;
                   "signalKVSStation".qManualMode.Conv_FRV[#i] := false;
               END_IF;


               //vibroTable
               IF "hmi".addedVibro.manStartVibroTable[#i] THEN
                   "signalKVSStation".qManualMode.vibroTable[#i] := true;
               ELSE
                   "signalKVSStation".qManualMode.vibroTable[#i] := false;
               END_IF;


           END_IF;

           // //flipper
           #flipper(openQ => "signalKVSStation".qManualMode.flipper_Up,
                    closeQ => "signalKVSStation".qManualMode.flipper_Down,
                    open := "hmi".plavnik.manOpenPlavnik,
                    close := "hmi".plavnik.manClosePlavnik,
                    "time_open/close" := t#250ms,
                    stopAlarm := #stopAlarm);
           //питатель
           IF "hmi".sourceConv.manStartConv THEN
               "signalKVSStation".qManualMode.startInConv := true;
           ELSE
               "signalKVSStation".qManualMode.startInConv := false;
           END_IF;

       ELSE
           //деактивируем сигналы на катушки ручного режима и
           //сигналы управления в ручном режиме
           "hmi".weightLine[#i].manOpenLeftValveWeightPocket := false;
           "signalKVSStation".qManualMode.Bunker_leftOpen[#i] := false;

           "hmi".weightLine[#i].manCloseLeftValveWeightPocket := false;
           "signalKVSStation".qManualMode.Bunker_leftClose[#i] := false;

           "hmi".weightLine[#i].manOpenRightValveWeightPocket := false;
           "signalKVSStation".qManualMode.Bunker_rightOpen[#i] := false;

           "hmi".weightLine[#i].manCloseRightValveWieghtPocket := false;
           "signalKVSStation".qManualMode.Bunker_rightClose[#i] := false;

           "hmi".weightLine[#i].manOpenRightValveWeightPocket := false;
           "signalKVSStation".qManualMode.Door_open[#i] := false;

           "hmi".weightLine[#i].manCloseValveAfterVibroLot := false;
           "signalKVSStation".qManualMode.Door_close[#i] := false;

           "hmi".weightLine[#i].manVibroLotStart := false;
           "signalKVSStation".qManualMode.vibroLot[#i] := false;
           IF #i = 1 OR #i = 2 THEN
               "hmi".outConvAndPack[#i].manStartOutConv := false;
               "signalKVSStation".qManualMode.Conv_FRV[#i] := false;
               "signalKVSStation".qManualMode.Conv_REV[#i] := false;

               "hmi".addedVibro.manStartVibroTable[#i] := false;
               "signalKVSStation".qManualMode.vibroTable[#i] := false;
           END_IF;
           "hmi".plavnik.manOpenPlavnik := false;
           "signalKVSStation".qManualMode.flipper_Up := false;

           "hmi".plavnik.manClosePlavnik := false;
           "signalKVSStation".qManualMode.flipper_Down := false;

           "hmi".sourceConv.manStartConv := false;
           "signalKVSStation".qManualMode.startInConv := false;



       END_IF;
   END_FOR;
END_REGION

REGION Network 3 (SCL): Части программы которые запускают сразу все однотипные узлы
   //запустить и остановить все вибролотки
   //
   #i := 0;
   FOR #i := 1 TO 12 DO
       IF "hmi".manRunAllVibroLot THEN
           "hmi".weightLine[#i].manVibroLotStart := true;
       END_IF;
       IF "hmi".manStopAllVibroLot THEN
           "hmi".weightLine[#i].manVibroLotStart := false;
       END_IF;
   END_FOR;
END_REGION
END_FUNCTION_BLOCK

FUNCTION_BLOCK "controlValve"   // FB2, LAD
{ S7_Optimized_Access := 'TRUE' }
VERSION : 0.1
// stored: AutoNumber true, IsIECCheckEnabled false, IsRetainMemResEnabled false, MemoryReserve 100, SetENOAutomatically false, UDAEnableTagReadback false
   VAR_INPUT
      autoclose_M : Bool;   // режим автозакрытия
      time_autoclose : Time := T#2000ms;
      "time_open/close" : Time := T#2000ms;
   END_VAR
   VAR_OUTPUT
      openQ : Bool;   // катушка на открытие
      closeQ : Bool;   // катушка на закрытие
   END_VAR
   VAR_IN_OUT
      open : Bool;   // сигнал на открытие
      close : Bool;   // сигнал на закрытие
      stopAlarm : Bool;   // сигнал резкого выключения
   END_VAR
   VAR
      tofOpen : TOF_TIME;   // время в течении которого катушка на открытие включена
      tofClose : TOF_TIME;   // время в течении которого катушка на закрытие включена
      Ptrig : Array[0..1] of Bool;   // триггеры ловят импульсный сигнал о включении и выключении
      Ntrig : Array[0..1] of Bool;
      tonAutoclose_M : TON_TIME;   // время через которое сработает автозакрытие
   END_VAR
   VAR_TEMP   // added for the SCL form of the ladder/FBD networks
      _w1 : Bool;
      _w2 : Bool;
      _w3 : Bool;
      _w4 : Bool;
      _w5 : Bool;
      _w6 : Bool;
   END_VAR
BEGIN

REGION Network 1: сигнал на открытие
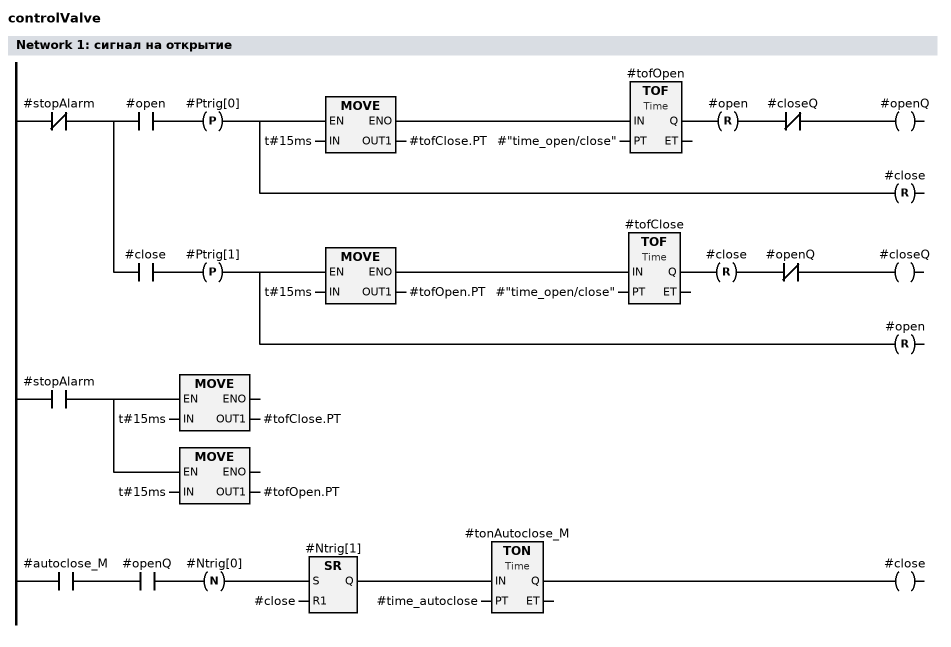
   RUNG wire#powerrail
      I_Contact( #stopAlarm )
      wire#w1
      Contact( #open )
      P_Trig( #Ptrig[0] )
      wire#w2
      Move(in := t#15ms, out1 => #tofClose.PT)
      { S7_Templates := "time_type := Time" } #tofOpen.TOF(pt := #"time_open/close", et =>)
      R_Coil( #open )
      I_Contact( #closeQ )
      Coil( #openQ )
   END_RUNG
   RUNG wire#w2
      R_Coil( #close )
   END_RUNG
   RUNG wire#w1
      Contact( #close )
      P_Trig( #Ptrig[1] )
      wire#w3
      Move(in := t#15ms, out1 => #tofOpen.PT)
      { S7_Templates := "time_type := Time" } #tofClose.TOF(pt := #"time_open/close", et =>)
      R_Coil( #close )
      I_Contact( #openQ )
      Coil( #closeQ )
   END_RUNG
   RUNG wire#w3
      R_Coil( #open )
   END_RUNG
   RUNG wire#powerrail
      Contact( #stopAlarm )
      wire#w4
      Move(in := t#15ms, out1 => #tofClose.PT)
   END_RUNG
   RUNG wire#w4
      Move(in := t#15ms, out1 => #tofOpen.PT)
   END_RUNG
   RUNG wire#powerrail
      Contact( #autoclose_M )
      Contact( #openQ )
      N_Trig( #Ntrig[0] )
      S_SR(operand := #Ntrig[1], r1 := #close)
      { S7_Templates := "time_type := Time" } #tonAutoclose_M.TON(pt := #time_autoclose, et =>)
      Coil( #close )
   END_RUNG
   // the same network as SCL:
   #_w1 := NOT #stopAlarm AND #open;
   #_w2 := #_w1 AND NOT #Ptrig[0];   // rising edge
   #Ptrig[0] := #_w1;
   IF #_w2 THEN #tofClose.PT := t#15ms; END_IF;
   #tofOpen(IN := #_w2, PT := #"time_open/close");   // TOF
   IF #tofOpen.Q THEN #open := FALSE; END_IF;
   #openQ := #tofOpen.Q AND NOT #closeQ;
   IF #_w2 THEN #close := FALSE; END_IF;
   #_w3 := NOT #stopAlarm AND #close;
   #_w4 := #_w3 AND NOT #Ptrig[1];   // rising edge
   #Ptrig[1] := #_w3;
   IF #_w4 THEN #tofOpen.PT := t#15ms; END_IF;
   #tofClose(IN := #_w4, PT := #"time_open/close");   // TOF
   IF #tofClose.Q THEN #close := FALSE; END_IF;
   #closeQ := #tofClose.Q AND NOT #openQ;
   IF #_w4 THEN #open := FALSE; END_IF;
   IF #stopAlarm THEN
       #tofClose.PT := t#15ms;
       #tofOpen.PT := t#15ms;
   END_IF;
   #_w5 := #autoclose_M AND #openQ;
   #_w6 := NOT #_w5 AND #Ntrig[0];   // falling edge
   #Ntrig[0] := #_w5;
   IF #_w6 THEN
       #Ntrig[1] := TRUE;   // SR flip-flop
   END_IF;
   IF #close THEN #Ntrig[1] := FALSE; END_IF;
   #tonAutoclose_M(IN := #Ntrig[1], PT := #time_autoclose);   // TON
   #close := #tonAutoclose_M.Q;
END_REGION
END_FUNCTION_BLOCK

FUNCTION_BLOCK "AutoMode"   // FB20, LAD
TITLE = Автоматический режим
{ S7_Optimized_Access := 'TRUE' }
VERSION : 0.1
// //setWeight - уставка веса в упаковке => используется при подсчете уставок в бункера
// //speed_inConveyer - уставка скорости на питателе в %
// //speedVibro - уставка скорости вибрации в %
// //maxWeightBunker - максимальный вес в один бункер => используется при подсчете уставок в бункера
// //workPlavnik - использовать ли плавник во время работы 
// //measurementError - допустимая погрешность на итоговый вес => используется при поиске подходящих бункеров при сбросе
// //mediumWeightProduct - средний вес продукта => используется при подсчете уставок в бункера
// stored: AutoNumber false, IsIECCheckEnabled false, IsRetainMemResEnabled false, MemoryReserve 100, SetENOAutomatically false, UDAEnableTagReadback false
   VAR_IN_OUT
      enableAutoMode : Bool;   // разрешение на переход в автоматический режим
      isFinishPreWork : Bool;   // сигнал об окончании подготовки к автоматическому режиму
      isStartAutoMode : Bool;   // сигнал что автоматический режим запущен
   END_VAR
   VAR
      TaskSetWeight : Real;   // целевой вес который ищем в сортировке
      SetWeightBunker : Array[0..12] of Real;   // уставки весов в бункера
      currentWeightBunker : Array[0..12] of Real;
      readyToSort : Array[0..12] of Bool;   // массив говорящий какие бункера готовы к сортировке
      readyToDrop : Array[0..12] of Bool;   // массив говорящий какие бункера надо сбросить
      readyToDropYP : Array[0..2] of Bool;
      isWorkWithBunker : Array[0..12] of Bool;   // массив разрешающий бункерам работать
      preWorkAutoMode : Struct
         isFinishPreWork : Bool;
         alarmStop : Bool;
      END_STRUCT;
      preWork_AM_FB : "preWork_AM";
      workPackingMachine_AM_FB : "workPackingMachine_AM";
      workInConveyer_AM_FB : "workInConveyer_AM";
      controlFllipper_AM_FB : "controlValve";
      workVibroLot_AM_FB : Array[0..12] of "workVibroLot_AM";
      workVibroTable_AM_FB : "workVibroTable_AM";
      weightModule_AM_FB : "weightModule_AM";
      Sorting_AM_FB : "Sorting_AM";
      setWeightBunker_FB : "setWeightBunker_AM";
      blockSorting : Bool;   // запрет на сортировку в блоке сортировке
      openFlipper : Bool;
      hmiYpDropWeight : Array[0..2] of Real;
      hmiYpDropError : Array[0..2] of Real;
   END_VAR
   VAR_TEMP
      "!!!!!" : Array[0..1] of Bool;
      i : DInt;
      tmpStableWeightBunker : Array[0..12] of Real;
   END_VAR
BEGIN

REGION Network 1: Аварийный останов
   // По нажатию кнопки Стоп и Аварийный стоп
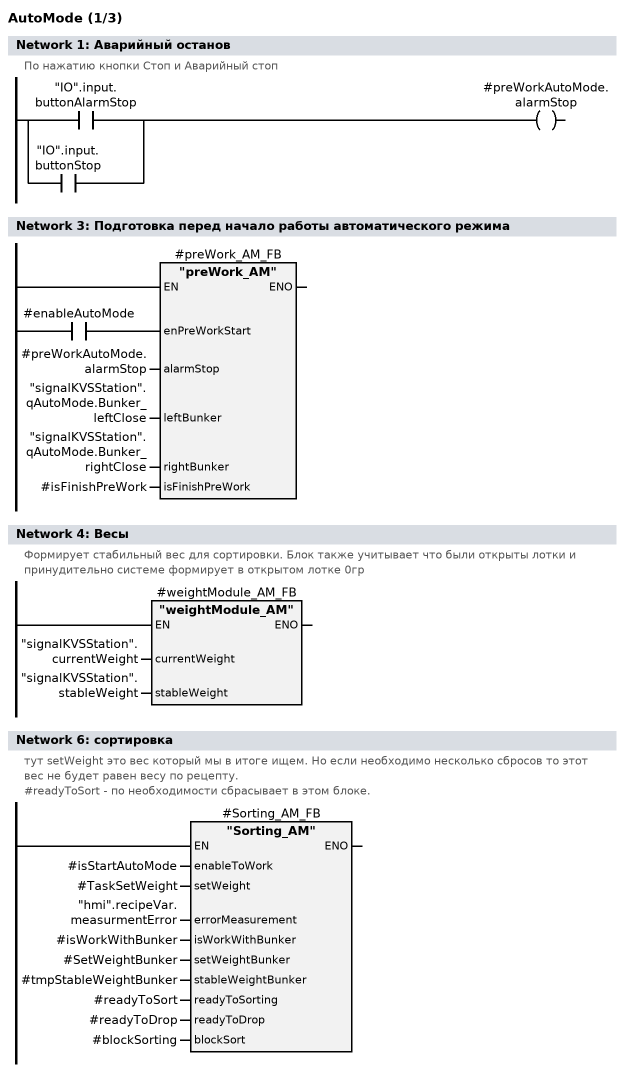
   RUNG wire#powerrail
      Contact( "IO".input.buttonAlarmStop )
      wire#w1
      Coil( #preWorkAutoMode.alarmStop )
   END_RUNG
   RUNG wire#powerrail
      Contact( "IO".input.buttonStop )
   END_RUNG wire#w1
   // the same network as SCL:
   #preWorkAutoMode.alarmStop := "IO".input.buttonAlarmStop OR "IO".input.buttonStop;
END_REGION

REGION Network 2 (SCL): статусы автоматического режима
   IF #enableAutoMode THEN
       IF NOT (#isFinishPreWork) THEN
           "hmi".readySystem := 2;
       ELSE
           IF NOT (#isStartAutoMode) THEN
               "hmi".readySystem := 0;
           ELSE
               "hmi".readySystem := 1;
           END_IF;
       END_IF;
   END_IF;
END_REGION

REGION Network 3: Подготовка перед начало работы автоматического режима
   RUNG wire#powerrail
      #preWork_AM_FB(enPreWorkStart := wire#w1, alarmStop := #preWorkAutoMode.alarmStop, leftBunker := "signalKVSStation".qAutoMode.Bunker_leftClose, rightBunker := "signalKVSStation".qAutoMode.Bunker_rightClose, isFinishPreWork := #isFinishPreWork)
   END_RUNG
   RUNG wire#powerrail
      Contact( #enableAutoMode )
   END_RUNG wire#w1
   // the same network as SCL:
   #preWork_AM_FB(enPreWorkStart := #enableAutoMode,   // "preWork_AM"
                  alarmStop := #preWorkAutoMode.alarmStop,
                  leftBunker := "signalKVSStation".qAutoMode.Bunker_leftClose,
                  rightBunker := "signalKVSStation".qAutoMode.Bunker_rightClose,
                  isFinishPreWork := #isFinishPreWork);
END_REGION

REGION Network 4: Весы
   // Формирует стабильный вес для сортировки. Блок также учитывает что были открыты лотки и принудительно системе формирует в открытом лотке 0гр
   RUNG wire#powerrail
      #weightModule_AM_FB(currentWeight := "signalKVSStation".currentWeight, stableWeight := "signalKVSStation".stableWeight)
   END_RUNG
   // the same network as SCL:
   #weightModule_AM_FB(currentWeight := "signalKVSStation".currentWeight,   // "weightModule_AM"
                       stableWeight := "signalKVSStation".stableWeight);
END_REGION

REGION Network 5 (SCL): выделяем стабильные веса с которыми будем работать
   #i := 0;
   FOR #i := 1 TO 12 DO
       #tmpStableWeightBunker[#i] := "signalKVSStation".stableWeight[#i].weight[0];
       "hmi".weightLine[#i].currentWeightPocket := "signalKVSStation".stableWeight[#i].weight[0];
       "hmi".weightLine[#i].targetWeightPocket := #SetWeightBunker[#i];
   END_FOR;
   #currentWeightBunker := "signalKVSStation".currentWeight;
END_REGION

REGION Network 6: сортировка
   // тут setWeight это вес который мы в итоге ищем. Но если необходимо несколько сбросов то этот вес не будет равен весу по рецепту.
   // #readyToSort - по необходимости сбрасывает в этом блоке.
   RUNG wire#powerrail
      #Sorting_AM_FB(enableToWork := #isStartAutoMode, setWeight := #TaskSetWeight, errorMeasurement := "hmi".recipeVar.measurmentError, isWorkWithBunker := #isWorkWithBunker, setWeightBunker := #SetWeightBunker, stableWeightBunker := #tmpStableWeightBunker, readyToSorting := #readyToSort, readyToDrop := #readyToDrop, blockSort := #blockSorting)
   END_RUNG
   // the same network as SCL:
   #Sorting_AM_FB(enableToWork := #isStartAutoMode,   // "Sorting_AM"
                  setWeight := #TaskSetWeight,
                  errorMeasurement := "hmi".recipeVar.measurmentError,
                  isWorkWithBunker := #isWorkWithBunker,
                  setWeightBunker := #SetWeightBunker,
                  stableWeightBunker := #tmpStableWeightBunker,
                  readyToSorting := #readyToSort,
                  readyToDrop := #readyToDrop,
                  blockSort := #blockSorting);
END_REGION

REGION Network 7 (SCL): Перенос данных для панели
   "hmi".permitOn1Bunk := "hmi".permitOn2Bunk := #readyToDrop;
END_REGION

REGION Network 8: Расчет уставок в бункере
   // Здесь происходит расчет уставок на все бункера в зависимости от: веса уставки, максимального веса в один бункер, среднего веса продукта
   // Также управление конвейерами, упаковочными машинами и бункерами
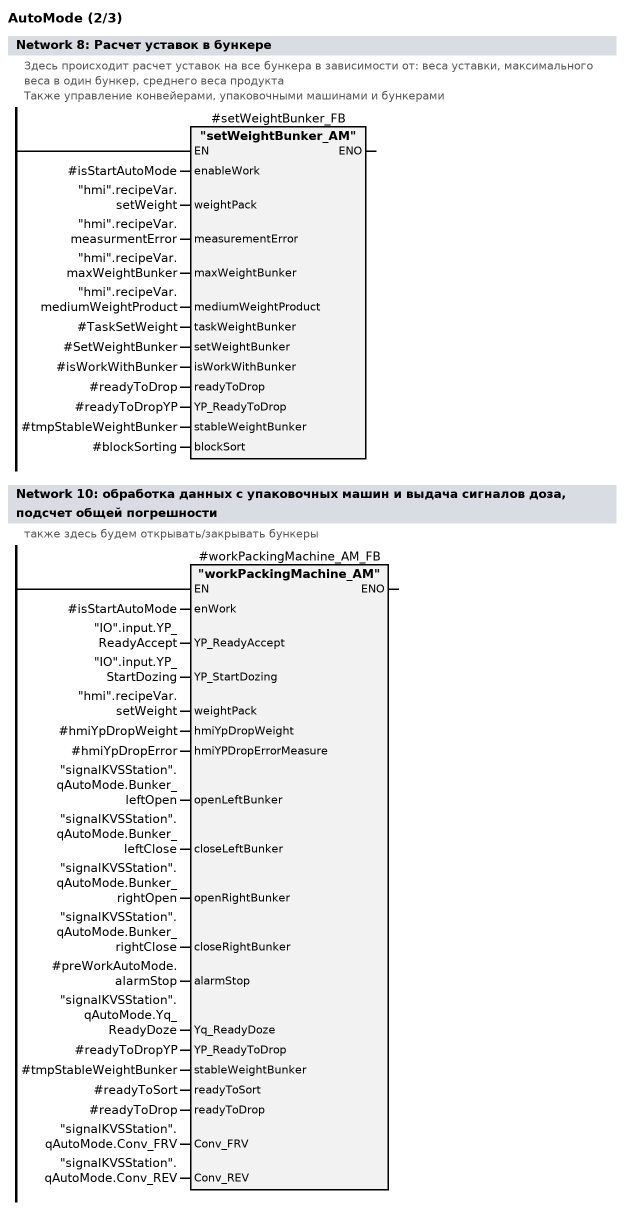
   RUNG wire#powerrail
      #setWeightBunker_FB(enableWork := #isStartAutoMode, weightPack := "hmi".recipeVar.setWeight, measurementError := "hmi".recipeVar.measurmentError, maxWeightBunker := "hmi".recipeVar.maxWeightBunker, mediumWeightProduct := "hmi".recipeVar.mediumWeightProduct, taskWeightBunker := #TaskSetWeight, setWeightBunker := #SetWeightBunker, isWorkWithBunker := #isWorkWithBunker, readyToDrop := #readyToDrop, YP_ReadyToDrop := #readyToDropYP, stableWeightBunker := #tmpStableWeightBunker, blockSort := #blockSorting)
   END_RUNG
   // the same network as SCL:
   #setWeightBunker_FB(enableWork := #isStartAutoMode,   // "setWeightBunker_AM"
                       weightPack := "hmi".recipeVar.setWeight,
                       measurementError := "hmi".recipeVar.measurmentError,
                       maxWeightBunker := "hmi".recipeVar.maxWeightBunker,
                       mediumWeightProduct := "hmi".recipeVar.mediumWeightProduct,
                       taskWeightBunker := #TaskSetWeight,
                       setWeightBunker := #SetWeightBunker,
                       isWorkWithBunker := #isWorkWithBunker,
                       readyToDrop := #readyToDrop,
                       YP_ReadyToDrop := #readyToDropYP,
                       stableWeightBunker := #tmpStableWeightBunker,
                       blockSort := #blockSorting);
END_REGION

REGION Network 9 (SCL): передача уставок в панель
   #i := 0;
   FOR #i := 1 TO 12 DO
       "hmi".weightLine[#i].targetWeightPocket := #SetWeightBunker[#i];
   END_FOR;
END_REGION

REGION Network 10: обработка данных с упаковочных машин и выдача сигналов доза, подсчет общей погрешности
   // также здесь будем открывать/закрывать бункеры
   RUNG wire#powerrail
      #workPackingMachine_AM_FB(enWork := #isStartAutoMode, YP_ReadyAccept := "IO".input.YP_ReadyAccept, YP_StartDozing := "IO".input.YP_StartDozing, weightPack := "hmi".recipeVar.setWeight, hmiYpDropWeight := #hmiYpDropWeight, hmiYPDropErrorMeasure := #hmiYpDropError, openLeftBunker := "signalKVSStation".qAutoMode.Bunker_leftOpen, closeLeftBunker := "signalKVSStation".qAutoMode.Bunker_leftClose, openRightBunker := "signalKVSStation".qAutoMode.Bunker_rightOpen, closeRightBunker := "signalKVSStation".qAutoMode.Bunker_rightClose, alarmStop := #preWorkAutoMode.alarmStop, Yq_ReadyDoze := "signalKVSStation".qAutoMode.Yq_ReadyDoze, YP_ReadyToDrop := #readyToDropYP, stableWeightBunker := #tmpStableWeightBunker, readyToSort := #readyToSort, readyToDrop := #readyToDrop, Conv_FRV := "signalKVSStation".qAutoMode.Conv_FRV, Conv_REV := "signalKVSStation".qAutoMode.Conv_REV)
   END_RUNG
   // the same network as SCL:
   #workPackingMachine_AM_FB(enWork := #isStartAutoMode,   // "workPackingMachine_AM"
                           YP_ReadyAccept := "IO".input.YP_ReadyAccept,
                           YP_StartDozing := "IO".input.YP_StartDozing,
                           weightPack := "hmi".recipeVar.setWeight,
                           hmiYpDropWeight := #hmiYpDropWeight,
                           hmiYPDropErrorMeasure := #hmiYpDropError,
                           openLeftBunker := "signalKVSStation".qAutoMode.Bunker_leftOpen,
                           closeLeftBunker := "signalKVSStation".qAutoMode.Bunker_leftClose,
                           openRightBunker := "signalKVSStation".qAutoMode.Bunker_rightOpen,
                           closeRightBunker := "signalKVSStation".qAutoMode.Bunker_rightClose,
                           alarmStop := #preWorkAutoMode.alarmStop,
                           Yq_ReadyDoze := "signalKVSStation".qAutoMode.Yq_ReadyDoze,
                           YP_ReadyToDrop := #readyToDropYP,
                           stableWeightBunker := #tmpStableWeightBunker,
                           readyToSort := #readyToSort,
                           readyToDrop := #readyToDrop,
                           Conv_FRV := "signalKVSStation".qAutoMode.Conv_FRV,
                           Conv_REV := "signalKVSStation".qAutoMode.Conv_REV);
END_REGION

REGION Network 11 (SCL)
   #i := 0;
   FOR #i := 1 TO 2 DO
       "hmi".outConvAndPack[#i].currentWeightPack := #hmiYpDropWeight[#i];
       "hmi".outConvAndPack[#i].currentErrorMeasure := #hmiYpDropError[#i];
   END_FOR;
END_REGION

REGION Network 12: Работа конвейера
   // конвейер работает пока не сработал датчик пересыпа
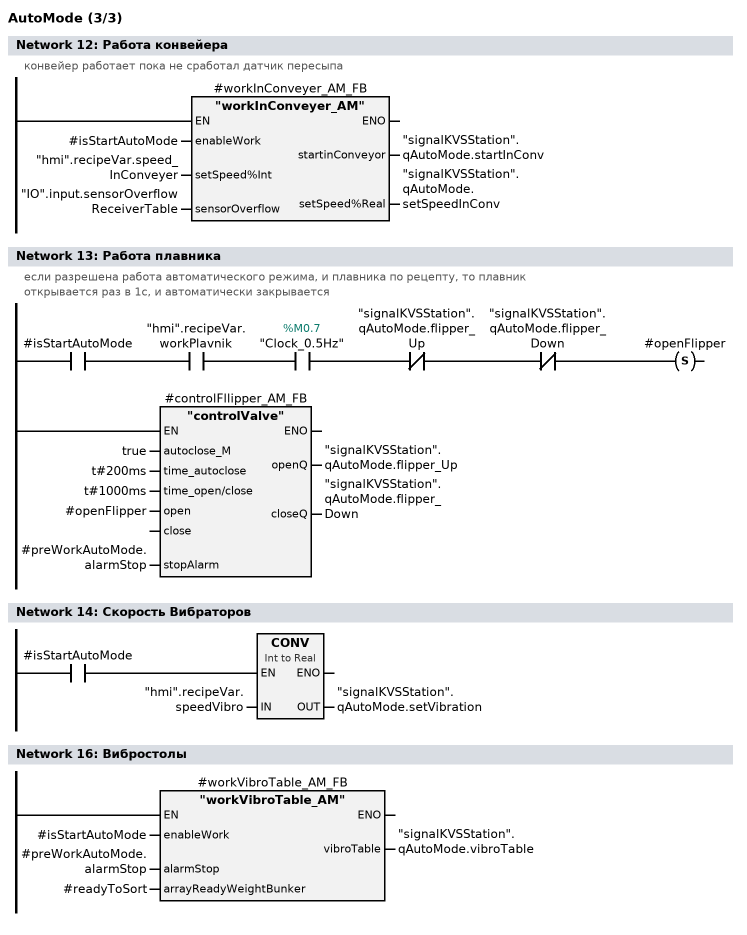
   RUNG wire#powerrail
      #workInConveyer_AM_FB(enableWork := #isStartAutoMode, "setSpeed%Int" := "hmi".recipeVar.speed_InConveyer, sensorOverflow := "IO".input.sensorOverflowReceiverTable, startinConveyor => "signalKVSStation".qAutoMode.startInConv, "setSpeed%Real" => "signalKVSStation".qAutoMode.setSpeedInConv)
   END_RUNG
   // the same network as SCL:
   #workInConveyer_AM_FB(enableWork := #isStartAutoMode,   // "workInConveyer_AM"
                         "setSpeed%Int" := "hmi".recipeVar.speed_InConveyer,
                         sensorOverflow := "IO".input.sensorOverflowReceiverTable,
                         startinConveyor => "signalKVSStation".qAutoMode.startInConv,
                         "setSpeed%Real" => "signalKVSStation".qAutoMode.setSpeedInConv);
END_REGION

REGION Network 13: Работа плавника
   // если разрешена работа автоматического режима, и плавника по рецепту, то плавник
   // открывается раз в 1с, и автоматически закрывается
   RUNG wire#powerrail
      Contact( #isStartAutoMode )
      Contact( "hmi".recipeVar.workPlavnik )
      Contact( "Clock_0.5Hz" )
      I_Contact( "signalKVSStation".qAutoMode.flipper_Up )
      I_Contact( "signalKVSStation".qAutoMode.flipper_Down )
      S_Coil( #openFlipper )
   END_RUNG
   RUNG wire#powerrail
      #controlFllipper_AM_FB(autoclose_M := true, time_autoclose := t#200ms, "time_open/close" := t#1000ms, open := #openFlipper, close :=, stopAlarm := #preWorkAutoMode.alarmStop, openQ => "signalKVSStation".qAutoMode.flipper_Up, closeQ => "signalKVSStation".qAutoMode.flipper_Down)
   END_RUNG
   // the same network as SCL:
   IF #isStartAutoMode AND "hmi".recipeVar.workPlavnik AND "Clock_0.5Hz" AND NOT "signalKVSStation".qAutoMode.flipper_Up AND NOT "signalKVSStation".qAutoMode.flipper_Down THEN
       #openFlipper := TRUE;
   END_IF;
   #controlFllipper_AM_FB(autoclose_M := true,   // "controlValve"
                          time_autoclose := t#200ms,
                          "time_open/close" := t#1000ms,
                          open := #openFlipper,
                          stopAlarm := #preWorkAutoMode.alarmStop,
                          openQ => "signalKVSStation".qAutoMode.flipper_Up,
                          closeQ => "signalKVSStation".qAutoMode.flipper_Down);
END_REGION

REGION Network 14: Скорость Вибраторов
   RUNG wire#powerrail
      Contact( #isStartAutoMode )
      { S7_Templates := "[SrcType := Int, DestType := Real]" } Convert(in := "hmi".recipeVar.speedVibro, out => "signalKVSStation".qAutoMode.setVibration)
   END_RUNG
   // the same network as SCL:
   IF #isStartAutoMode THEN
       "signalKVSStation".qAutoMode.setVibration := INT_TO_REAL("hmi".recipeVar.speedVibro);
   END_IF;
END_REGION

REGION Network 15 (SCL): Вибролотки, лопатки
   #i := 0;
   FOR #i := 1 TO 12 DO
       #workVibroLot_AM_FB[#i](enableWork := #isStartAutoMode,
                               setWeightBunker := #SetWeightBunker[#i],
                               currentWeight := #currentWeightBunker[#i],//"signalKVSStation".stableWeight[#i].weight[0],
                               stateDoor := "hmi".weightLine[#i].stateValveAfterVibroLot,
                               stateBunkerLeft:="hmi".weightLine[#i].stateLeftValveWeightPocket,
                               stateBunkerRight:="hmi".weightLine[#i].stateRightValveWeightPocket,
                               alarmStop := #preWorkAutoMode.alarmStop,
                               isWorkWithBunker := #isWorkWithBunker[#i],

                               onVibroLot:= "signalKVSStation".qAutoMode.vibroLot[#i],
                               openDoor := "signalKVSStation".qAutoMode.Door_open[#i],
                               closeDoor := "signalKVSStation".qAutoMode.Door_close[#i],

                               isReadyToDrop:=#readyToDrop[#i],
                               isReadyToSort := #readyToSort[#i]);

   END_FOR;
END_REGION

REGION Network 16: Вибростолы
   RUNG wire#powerrail
      #workVibroTable_AM_FB(enableWork := #isStartAutoMode, alarmStop := #preWorkAutoMode.alarmStop, arrayReadyWeightBunker := #readyToSort, vibroTable => "signalKVSStation".qAutoMode.vibroTable)
   END_RUNG
   // the same network as SCL:
   #workVibroTable_AM_FB(enableWork := #isStartAutoMode,   // "workVibroTable_AM"
                         alarmStop := #preWorkAutoMode.alarmStop,
                         arrayReadyWeightBunker := #readyToSort,
                         vibroTable => "signalKVSStation".qAutoMode.vibroTable);
END_REGION
END_FUNCTION_BLOCK

FUNCTION_BLOCK "preWork_AM"   // FB5, LAD
{ S7_Optimized_Access := 'TRUE' }
VERSION : 0.1
// stored: AutoNumber true, IsIECCheckEnabled false, IsRetainMemResEnabled false, MemoryReserve 100, SetENOAutomatically false, UDAEnableTagReadback false
   VAR_INPUT
      enPreWorkStart : Bool;   // начало пред подготовки
   END_VAR
   VAR_IN_OUT
      alarmStop { ExternalAccessible := 'False'; ExternalVisible := 'False'; ExternalWritable := 'False'} : Bool;   // если пришел аварийный останов
      leftBunker : Array[0..12] of Bool;   // массив закрыть левые бункеры
      rightBunker : Array[0..12] of Bool;   // массив закрыть правые бункеры
      isFinishPreWork : Bool;   // сигнал о окончании подготовки автоматического режима
   END_VAR
   VAR
      closeLeftBunker_FB : Array[0..12] of "controlValve";
      closeRightBunker_FB : Array[0..12] of "controlValve";
      tempButtonLeft : Array[0..12] of Bool;
      tempButtonRight : Array[0..12] of Bool;
      valueControlBit : Bool;
      watchQ : Bool;
      tmpControlValue : Bool;
      tempP_trig : Array[0..1] of Bool;
   END_VAR
   VAR_TEMP
      i : DInt;
   END_VAR
   VAR_TEMP   // added for the SCL form of the ladder/FBD networks
      _w1 : Bool;
      _w2 : Bool;
   END_VAR
BEGIN

REGION Network 1
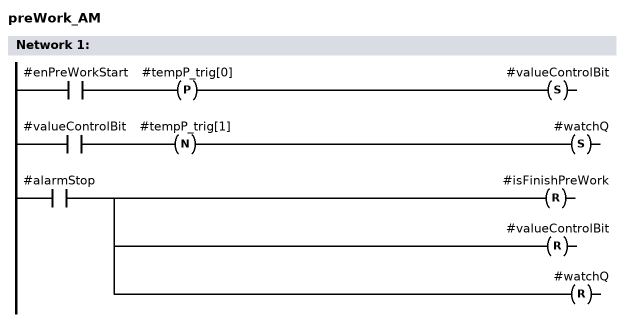
   RUNG wire#powerrail
      Contact( #enPreWorkStart )
      P_Trig( #tempP_trig[0] )
      S_Coil( #valueControlBit )
   END_RUNG
   RUNG wire#powerrail
      Contact( #valueControlBit )
      N_Trig( #tempP_trig[1] )
      S_Coil( #watchQ )
   END_RUNG
   RUNG wire#powerrail
      Contact( #alarmStop )
      wire#w1
      R_Coil( #isFinishPreWork )
   END_RUNG
   RUNG wire#w1
      R_Coil( #valueControlBit )
   END_RUNG
   RUNG wire#w1
      R_Coil( #watchQ )
   END_RUNG
   // the same network as SCL:
   #_w1 := #enPreWorkStart AND NOT #tempP_trig[0];   // rising edge
   #tempP_trig[0] := #enPreWorkStart;
   IF #_w1 THEN #valueControlBit := TRUE; END_IF;
   #_w2 := NOT #valueControlBit AND #tempP_trig[1];   // falling edge
   #tempP_trig[1] := #valueControlBit;
   IF #_w2 THEN #watchQ := TRUE; END_IF;
   IF #alarmStop THEN
       #isFinishPreWork := FALSE;
       #valueControlBit := FALSE;
       #watchQ := FALSE;
   END_IF;
END_REGION

REGION Network 2 (SCL)
       //если нет допуска то нет и разрешения на проверку
       //
       IF NOT (#enPreWorkStart) THEN
           #valueControlBit := false;
           #watchQ := false;
           #isFinishPreWork := false;
       END_IF;

       //проверка(выдержка) пока все закроются
       IF #watchQ THEN
           #i := 0;
           #tmpControlValue := true;
           FOR #i := 1 TO 12 DO
               #tmpControlValue := #tmpControlValue AND NOT (#closeLeftBunker_FB[#i].closeQ);
               #tmpControlValue := #tmpControlValue AND NOT (#closeRightBunker_FB[#i].closeQ);
           END_FOR;
           IF #tmpControlValue THEN//как только все закрыто то проверка закончена
               #watchQ := false;
               #isFinishPreWork := true;
           END_IF;
       END_IF;


       //управление механизмом закрытия
       IF NOT(#isFinishPreWork) THEN
           #i := 0;
           FOR #i := 1 TO 12 DO
               #tempButtonLeft[#i] :=#tempButtonRight[#i] := #valueControlBit;
               #closeLeftBunker_FB[#i](closeQ => #leftBunker[#i],
                                       close := #tempButtonLeft[#i],
                                       stopAlarm := #alarmStop,
                                       "time_open/close":=t#200ms);

               #closeRightBunker_FB[#i](closeQ => #rightBunker[#i],
                                        close := #tempButtonRight[#i],
                                        stopAlarm := #alarmStop,
                                        "time_open/close":=t#200ms);
           END_FOR;
           IF #valueControlBit THEN//сбрасываем бит на закрытие
               #valueControlBit := false;
           END_IF;
       END_IF;
END_REGION
END_FUNCTION_BLOCK

FUNCTION_BLOCK "weightModule_AM"   // FB12, LAD
{ S7_Optimized_Access := 'TRUE' }
VERSION : 0.1
// stored: AutoNumber true, IsIECCheckEnabled false, IsRetainMemResEnabled false, MemoryReserve 100, SetENOAutomatically false, UDAEnableTagReadback false
   VAR_IN_OUT
      currentWeight : Array[0..12] of Real;   // текущий вес
      stableWeight : Array[0..12] of "stableWeight";   // массивы стабильных весов
   END_VAR
   VAR
      tonSetStableWeight : Array[0..12] of TON_TIME;   // выдержка для переноса текущего веса в разряд стабильных
      prevWeight : Array[0..12] of Real;   // предыдущий вес
      runTaimerStableWeight : Array[0..12] of Bool;
      RS_TRIG_openBunker : Array[0..12] of Bool;   // триггер что бункера были открыты
   END_VAR
   VAR_TEMP
      i : DInt;
   END_VAR
BEGIN

REGION Network 1 (SCL)
   #i := 0;
   FOR #i := 1 TO 12 DO

       IF "hmi".weightLine[#i].stateLeftValveWeightPocket OR "hmi".weightLine[#i].stateRightValveWeightPocket THEN
           #RS_TRIG_openBunker[#i] := true;//фиксируем что произошло открытие бункеров
       END_IF;
       IF NOT("hmi".weightLine[#i].stateLeftValveWeightPocket) AND NOT("hmi".weightLine[#i].stateRightValveWeightPocket) THEN
           #RS_TRIG_openBunker[#i] := false;//если бункера закрыты, то сбрасываем фиксацию о их открытии
       END_IF;

       IF NOT (#RS_TRIG_openBunker[#i]) THEN

           IF (#prevWeight[#i] - 10) <= #currentWeight[#i] AND #currentWeight[#i] <= (#prevWeight[#i] + 10) THEN
               #runTaimerStableWeight[#i] := true;
           ELSE
               #runTaimerStableWeight[#i] := false;
               #prevWeight[#i] := #currentWeight[#i];
           END_IF;

